DATA_BLOCK "DO_1_2_TON"   // DB244
{ S7_Optimized_Access := 'TRUE' }
AUTHOR : Simatic
FAMILY : IEC
NAME : IEC_TMR
VERSION : 1.0
// stored: InstanceOfName IEC_TIMER
"IEC_TIMER"
BEGIN
END_DATA_BLOCK

DATA_BLOCK "DO_2_0_TOF"   // DB246
{ S7_Optimized_Access := 'TRUE' }
AUTHOR : Simatic
FAMILY : IEC
NAME : IEC_TMR
VERSION : 1.0
// stored: InstanceOfName IEC_TIMER
"IEC_TIMER"
BEGIN
END_DATA_BLOCK

DATA_BLOCK "DO_1_2_TOF"   // DB247
{ S7_Optimized_Access := 'TRUE' }
AUTHOR : Simatic
FAMILY : IEC
NAME : IEC_TMR
VERSION : 1.0
// stored: InstanceOfName IEC_TIMER
"IEC_TIMER"
BEGIN
END_DATA_BLOCK

DATA_BLOCK "DI_1_1_TOF"   // DB253
{ S7_Optimized_Access := 'TRUE' }
AUTHOR : Simatic
FAMILY : IEC
NAME : IEC_TMR
VERSION : 1.0
// stored: InstanceOfName IEC_TIMER
"IEC_TIMER"
BEGIN
END_DATA_BLOCK

DATA_BLOCK "DI_1_4_TOF"   // DB255
{ S7_Optimized_Access := 'TRUE' }
AUTHOR : Simatic
FAMILY : IEC
NAME : IEC_TMR
VERSION : 1.0
// stored: InstanceOfName IEC_TIMER
"IEC_TIMER"
BEGIN
END_DATA_BLOCK

DATA_BLOCK "DI_1_11_TOF"   // DB256
{ S7_Optimized_Access := 'TRUE' }
AUTHOR : Simatic
FAMILY : IEC
NAME : IEC_TMR
VERSION : 1.0
// stored: InstanceOfName IEC_TIMER
"IEC_TIMER"
BEGIN
END_DATA_BLOCK

DATA_BLOCK "DO_1_4_TON"   // DB259
{ S7_Optimized_Access := 'TRUE' }
AUTHOR : Simatic
FAMILY : IEC
NAME : IEC_TMR
VERSION : 1.0
// stored: InstanceOfName IEC_TIMER
"IEC_TIMER"
BEGIN
END_DATA_BLOCK

DATA_BLOCK "DO_1_4_TOF"   // DB262
{ S7_Optimized_Access := 'TRUE' }
AUTHOR : Simatic
FAMILY : IEC
NAME : IEC_TMR
VERSION : 1.0
// stored: InstanceOfName IEC_TIMER
"IEC_TIMER"
BEGIN
END_DATA_BLOCK

DATA_BLOCK "DI_1_6_TOF"   // DB270
{ S7_Optimized_Access := 'TRUE' }
AUTHOR : Simatic
FAMILY : IEC
NAME : IEC_TMR
VERSION : 1.0
// stored: InstanceOfName IEC_TIMER
"IEC_TIMER"
BEGIN
END_DATA_BLOCK

DATA_BLOCK "DI_1_13_TOF"   // DB271
{ S7_Optimized_Access := 'TRUE' }
AUTHOR : Simatic
FAMILY : IEC
NAME : IEC_TMR
VERSION : 1.0
// stored: InstanceOfName IEC_TIMER
"IEC_TIMER"
BEGIN
END_DATA_BLOCK

DATA_BLOCK "DO_1_6_TON"   // DB274
{ S7_Optimized_Access := 'TRUE' }
AUTHOR : Simatic
FAMILY : IEC
NAME : IEC_TMR
VERSION : 1.0
// stored: InstanceOfName IEC_TIMER
"IEC_TIMER"
BEGIN
END_DATA_BLOCK

DATA_BLOCK "DO_1_6_TOF"   // DB277
{ S7_Optimized_Access := 'TRUE' }
AUTHOR : Simatic
FAMILY : IEC
NAME : IEC_TMR
VERSION : 1.0
// stored: InstanceOfName IEC_TIMER
"IEC_TIMER"
BEGIN
END_DATA_BLOCK

DATA_BLOCK "DI_1_2_TOF"   // DB285
{ S7_Optimized_Access := 'TRUE' }
AUTHOR : Simatic
FAMILY : IEC
NAME : IEC_TMR
VERSION : 1.0
// stored: InstanceOfName IEC_TIMER
"IEC_TIMER"
BEGIN
END_DATA_BLOCK

DATA_BLOCK "DI_1_5_TOF"   // DB287
{ S7_Optimized_Access := 'TRUE' }
AUTHOR : Simatic
FAMILY : IEC
NAME : IEC_TMR
VERSION : 1.0
// stored: InstanceOfName IEC_TIMER
"IEC_TIMER"
BEGIN
END_DATA_BLOCK

DATA_BLOCK "DI_1_12_TOF"   // DB288
{ S7_Optimized_Access := 'TRUE' }
AUTHOR : Simatic
FAMILY : IEC
NAME : IEC_TMR
VERSION : 1.0
// stored: InstanceOfName IEC_TIMER
"IEC_TIMER"
BEGIN
END_DATA_BLOCK

DATA_BLOCK "DO_1_5_TON"   // DB291
{ S7_Optimized_Access := 'TRUE' }
AUTHOR : Simatic
FAMILY : IEC
NAME : IEC_TMR
VERSION : 1.0
// stored: InstanceOfName IEC_TIMER
"IEC_TIMER"
BEGIN
END_DATA_BLOCK

DATA_BLOCK "DO_1_5_TOF"   // DB294
{ S7_Optimized_Access := 'TRUE' }
AUTHOR : Simatic
FAMILY : IEC
NAME : IEC_TMR
VERSION : 1.0
// stored: InstanceOfName IEC_TIMER
"IEC_TIMER"
BEGIN
END_DATA_BLOCK

// folder: (top level)

FUNCTION "Valve" : Void   // FC1, SCL
{ S7_Optimized_Access := 'TRUE' }
VERSION : 0.1
   VAR_INPUT
      Valve_opening : Bool;
      Need_open : Bool;
   END_VAR
   VAR_OUTPUT
      CMD_Open_Out : Bool;
      Alarm_Out : Bool;
   END_VAR
   VAR_IN_OUT
      valve : Struct
         CMD_Open : Bool;   // Команда открыть
         CMD_Close : Bool;   // Команда закрыть
         CMD_ALRM_Stop : Bool;
         State : Word;
         State_INT : Int;
         Mode : Bool;   // 0-ручной, 1-авто
         Alarm : Word;
         bools : Word;
         RST_ALRM : Bool;
         CMD_Open_Out : Bool;   // управление открыть
         CMD_Close_Out : Bool;   // управление закрыть
      END_STRUCT;
      TIME_Opening : TON_TIME;
      TIME_Closing : TON_TIME;
   END_VAR
BEGIN
   IF (#valve.Alarm = 0) AND #Need_open
   THEN
       #valve.CMD_Open := 1;
   ELSE
       #valve.CMD_Open := 0;
   END_IF;


   IF #valve.Alarm = 0
   THEN
      #valve.CMD_Open_Out := #valve.CMD_Open;

   ELSE
      #valve.CMD_Open_Out := FALSE;

   END_IF;

   //формирование состояний
   (*#valve.State.%X3 := #Valve_opening;
   #valve.State.%X4 := NOT (#Valve_opening);*)

   IF #valve.Alarm.%X1 THEN
       #valve.State := 1;
   END_IF;
   IF #valve.Alarm.%X2 THEN
       #valve.State := 2;
   END_IF;
   IF #Valve_opening AND NOT (#valve.Alarm.%X1 OR #valve.Alarm.%X2) THEN
       #valve.State := 3;
   END_IF;
   IF NOT (#Valve_opening) AND NOT (#valve.Alarm.%X1 OR #valve.Alarm.%X2) THEN
       #valve.State := 4;
   END_IF;

   //аварии при открытии и закрытии
   #TIME_Opening.TON(IN := #valve.CMD_Open_Out AND NOT (#Valve_opening),
   PT := T#25s);
   IF #TIME_Opening.Q THEN
       #valve.Alarm.%X1 := TRUE;
   END_IF;
   (*#valve.State.%X1 := #valve.Alarm.%X1;*)

   #TIME_Closing.TON(IN := NOT #valve.CMD_Open_Out AND #Valve_opening,
   PT := T#25s);
   IF #TIME_Closing.Q THEN
       #valve.Alarm.%X2 := TRUE;
   END_IF;
   (*#valve.State.%X2 := #valve.Alarm.%X2;*)

   IF #valve.RST_ALRM THEN
       #valve.Alarm := 0;
       #valve.RST_ALRM := 0;
   END_IF;



   #CMD_Open_Out := #valve.CMD_Open_Out;

   IF #valve.Alarm <> 0
   THEN
       #Alarm_Out := 1;
   END_IF;
END_FUNCTION

FUNCTION "DI" : Void   // FC2, LAD
{ S7_Optimized_Access := 'TRUE' }
VERSION : 0.1
   VAR_INPUT
      Input : Bool;   // Входной сигнал
   END_VAR
   VAR_IN_OUT
      DI : Struct
         Time_ON : Int;   // Время перехода OFF->ON
         Time_OFF : Int;   // Время перехода ON->OFF
         Input : Bool;   // Значение с модуля
         Disable : Bool;   // Запрет обработки канала
         Invert : Bool;   // Инертирование канала
         Output : Bool;   // Значение канала для логики
      END_STRUCT;
      TON_Timer : IEC_TIMER;
      TOF_Timer : IEC_TIMER;
   END_VAR
   VAR_TEMP
      Time_ON_int : Time;
      Time_OFF_int : Time;
      et1 : Time;
      et2 : Time;
      trig_et : Bool;
   END_VAR
BEGIN

REGION Network 1: Конверация времени
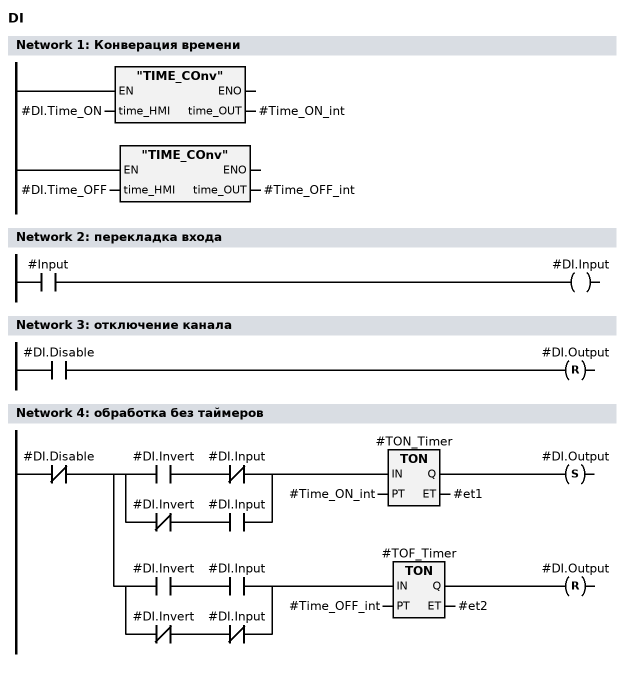
   RUNG wire#powerrail
      "TIME_COnv"(time_HMI := #DI.Time_ON, time_OUT => #Time_ON_int)
   END_RUNG
   RUNG wire#powerrail
      "TIME_COnv"(time_HMI := #DI.Time_OFF, time_OUT => #Time_OFF_int)
   END_RUNG
   // the same network as SCL:
   "TIME_COnv"(time_HMI := #DI.Time_ON, time_OUT => #Time_ON_int);
   "TIME_COnv"(time_HMI := #DI.Time_OFF, time_OUT => #Time_OFF_int);
END_REGION

REGION Network 2: перекладка входа
   RUNG wire#powerrail
      Contact( #Input )
      Coil( #DI.Input )
   END_RUNG
   // the same network as SCL:
   #DI.Input := #Input;
END_REGION

REGION Network 3: отключение канала
   RUNG wire#powerrail
      Contact( #DI.Disable )
      R_Coil( #DI.Output )
   END_RUNG
   // the same network as SCL:
   IF #DI.Disable THEN #DI.Output := FALSE; END_IF;
END_REGION

REGION Network 4: обработка без таймеров
   #TON_Timer.TON(IN := NOT #DI.Disable AND ((#DI.Invert AND NOT #DI.Input) OR (NOT #DI.Invert AND #DI.Input)),
                  PT := #Time_ON_int,
                  ET => #et1);
   IF #TON_Timer.Q THEN #DI.Output := TRUE; END_IF;
   #TOF_Timer.TON(IN := NOT #DI.Disable AND ((#DI.Invert AND #DI.Input) OR (NOT #DI.Invert AND NOT #DI.Input)),
                  PT := #Time_OFF_int,
                  ET => #et2);
   IF #TOF_Timer.Q THEN #DI.Output := FALSE; END_IF;
END_REGION
END_FUNCTION

FUNCTION "DO" : Void   // FC3, LAD
{ S7_Optimized_Access := 'TRUE' }
VERSION : 0.1
   VAR_OUTPUT
      Output : Bool;
   END_VAR
   VAR_IN_OUT
      "DO" : Struct
         Time_ON : Int;   // Время перехода OFF->ON
         Time_OFF : Int;   // Время перехода ON->OFF
         Input : Bool;   // Значение от логики
         Disable : Bool;   // Запрет обработки канала
         Invert : Bool;   // Инертирование канала
         Output : Bool;   // Значение на модуль
      END_STRUCT;
      TON_Timer : IEC_TIMER;
      TOF_Timer : IEC_TIMER;
   END_VAR
   VAR_TEMP
      Time_ON_int : Time;
      Time_OFF_int : Time;
      et1 : Time;
      et2 : Time;
   END_VAR
BEGIN

REGION Network 1: Конверация времени
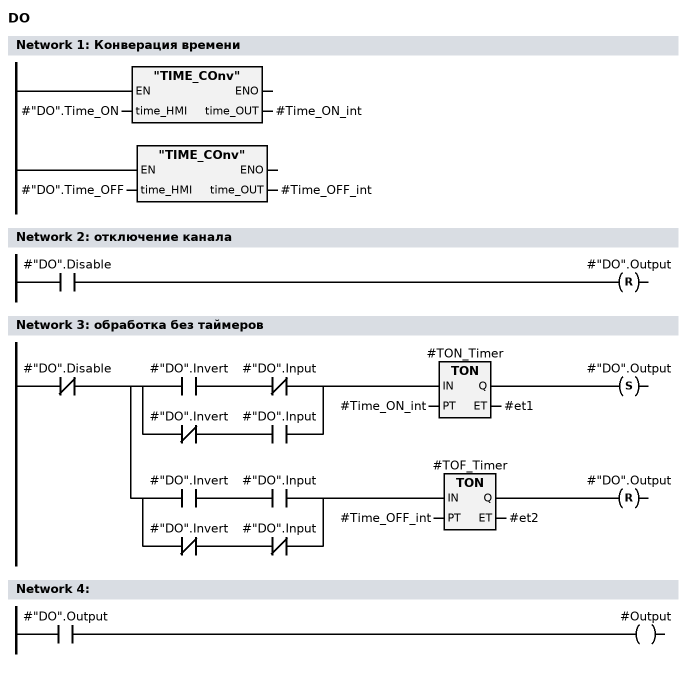
   RUNG wire#powerrail
      "TIME_COnv"(time_HMI := #"DO".Time_ON, time_OUT => #Time_ON_int)
   END_RUNG
   RUNG wire#powerrail
      "TIME_COnv"(time_HMI := #"DO".Time_OFF, time_OUT => #Time_OFF_int)
   END_RUNG
   // the same network as SCL:
   "TIME_COnv"(time_HMI := #"DO".Time_ON, time_OUT => #Time_ON_int);
   "TIME_COnv"(time_HMI := #"DO".Time_OFF, time_OUT => #Time_OFF_int);
END_REGION

REGION Network 2: отключение канала
   RUNG wire#powerrail
      Contact( #"DO".Disable )
      R_Coil( #"DO".Output )
   END_RUNG
   // the same network as SCL:
   IF #"DO".Disable THEN #"DO".Output := FALSE; END_IF;
END_REGION

REGION Network 3: обработка без таймеров
   #TON_Timer.TON(IN := NOT #"DO".Disable AND ((#"DO".Invert AND NOT #"DO".Input) OR (NOT #"DO".Invert AND #"DO".Input)),
                  PT := #Time_ON_int,
                  ET => #et1);
   IF #TON_Timer.Q THEN #"DO".Output := TRUE; END_IF;
   #TOF_Timer.TON(IN := NOT #"DO".Disable AND ((#"DO".Invert AND #"DO".Input) OR (NOT #"DO".Invert AND NOT #"DO".Input)),
                  PT := #Time_OFF_int,
                  ET => #et2);
   IF #TOF_Timer.Q THEN #"DO".Output := FALSE; END_IF;
END_REGION

REGION Network 4
   RUNG wire#powerrail
      Contact( #"DO".Output )
      Coil( #Output )
   END_RUNG
   // the same network as SCL:
   #Output := #"DO".Output;
END_REGION
END_FUNCTION

FUNCTION "Gaz" : Void   // FC4, SCL
{ S7_Optimized_Access := 'TRUE' }
VERSION : 0.1
BEGIN
   IF "PLC_Signals_DB".AI_2_6.State.%X1 THEN
       "DB_TST".Gaz_state := 2;
       ELSE 
           IF "PLC_Signals_DB".AI_2_6.State.%X2 THEN
               "DB_TST".Gaz_state := 1;
           ELSE
               "DB_TST".Gaz_state := 0;
           END_IF;
   END_IF;
END_FUNCTION

FUNCTION "AI_CONV" : Void   // FC6, SCL
{ S7_Optimized_Access := 'TRUE' }
VERSION : 0.1
   VAR_IN_OUT
      AI : Struct   // Структура AI
         Hihi_Value : Real;   // True
         High_Value : Real;   // True
         Low_Value : Real;   // True
         Lolo_Value : Real;   // True
         MIN_Current : Real;   // True
         MAX_Current : Real;   // True
         MAX_Value : Real;   // True
         MIN_Value : Real;   // True
         Underflow_RAW : Real;   // True
         Overflow_RAW : Real;   // True
         SCALED : Real;   // True
         ING_Value : Real;   // True
         Manual_Value : Real;   // True
         Alarm_Delay : Int;   // True
         Warning_Delay : Int;   // True
         AVG_Delay : Real;   // True
         Underflow_Delay : Int;   // True
         Overflow_Delay : Int;   // True
         State : Word;   // True
         Modeee : Word;   // True
         bools : Word;   // True
         AI_RAW_MIN : Int;   // True
         AI_RAW_MAX : Int;   // True
         Hihi_EN : Bool;   // True
         High_EN : Bool;   // True
         Low_En : Bool;   // True
         Lolo_EN : Bool;   // True
      END_STRUCT;
      AI_RAW : Int;   // ???????? ??? ?? ?????
      Hihi_TImer : TON_TIME;
      High_Timer : TON_TIME;
      Low_Timer : TON_TIME;
      Lolo_Timer : TON_TIME;
      WB_Timer : TON_TIME;
      OVerflow_Timer : TON_TIME;
   END_VAR
BEGIN
   (*
   #AI.mA := (#AI.ACP - #AI.ACP_LO) * ((#AI.mA_HI - #AI.mA_LO) / (#AI.ACP_HI - #AI.ACP_LO)) + #AI.mA_LO;
   #AI.ENG := (#AI.mA - #AI.mA_LO) * ((#AI.ENG_HI - #AI.ENG_LO) / (#AI.mA_HI - #AI.mA_LO)) + #AI.ENG_LO;
   *)
   //IF #AI.Modeee.%X0 THEN
       #AI.ING_Value := (#AI_RAW - #AI.AI_RAW_MIN) * ((#AI.MAX_Current - #AI.MIN_Current) / (#AI.AI_RAW_MAX - #AI.AI_RAW_MIN)) + #AI.MIN_Current;
       #AI.SCALED := (#AI_RAW - #AI.AI_RAW_MIN) * ((#AI.MAX_Value - #AI.MIN_Value) / (#AI.AI_RAW_MAX - #AI.AI_RAW_MIN)) + #AI.MIN_Value;




   //END_IF;


   (* #AI.mA := (#AI.ACP - #AI.ACP_LO) * ((#AI.mA_HI - #AI.mA_LO) / (#AI.ACP_HI - #AI.ACP_LO)) + #AI.mA_LO;
   #AI.ENG := (#AI.mA - #AI.mA_LO) * ((#AI.ENG_HI - #AI.ENG_LO) / (#AI.mA_HI - #AI.mA_LO)) + #AI.ENG_LO;

   IF NOT #AI.Repair THEN
       #AI.State_W.%X7 := FALSE;
       IF #AI.ENG <= #AI.ENG_Set_LoLo THEN
           #AI.LoLo := TRUE;
           #AI.State_W.%X0 := TRUE;
       ELSE
           #AI.LoLo := FALSE;
           #AI.State_W.%X0 := FALSE;
       END_IF;

       IF #AI.ENG <= #AI.ENG_Set_Lo THEN
           #AI.Lo := TRUE;
           #AI.State_W.%X1 := TRUE;
       ELSE
           #AI.Lo := FALSE;
           #AI.State_W.%X1 := FALSE;
       END_IF;

       IF #AI.ENG >= #AI.ENG_Set_Hi THEN
           #AI.Hi := TRUE;
           #AI.State_W.%X2 := TRUE;
       ELSE
           #AI.Hi := FALSE;
           #AI.State_W.%X2 := FALSE;
       END_IF;

       IF #AI.ENG >= #AI.ENG_Set_HiHi THEN
           #AI.HiHi := TRUE;
           #AI.State_W.%X3 := TRUE;
       ELSE
           #AI.HiHi := FALSE;
           #AI.State_W.%X3 := FALSE;
       END_IF;

       IF #AI.mA <= 3.5 THEN
           #AI.BL := TRUE;
           #AI.State_W.%X4 := TRUE;
       ELSE
           #AI.BL := FALSE;
           #AI.State_W.%X4 := FALSE;
       END_IF;

       IF #AI.mA >= 20.5 THEN
           #AI.OL := TRUE;
           #AI.State_W.%X5 := TRUE;
       ELSE
           #AI.OL := FALSE;
           #AI.State_W.%X5 := FALSE;
       END_IF;

       #AI.State_W.%X6 := #AI.State_W.%X4 OR #AI.State_W.%X5;

       IF #AI.OL OR #AI.BL THEN
           #AI.State := 3;
       ELSIF #AI.HiHi OR #AI.LoLo THEN
           #AI.State := 2;
       ELSIF #AI.Hi OR #AI.Lo THEN
           #AI.State := 1;
       ELSE
           #AI.State := 0;
       END_IF;

   ELSE
       #AI.LoLo := FALSE; #AI.Lo := FALSE; #AI.Hi := FALSE; #AI.HiHi := FALSE;
       #AI.OL := FALSE; #AI.BL := FALSE;
       #AI.State := 4;
       #AI.State_W := 0;
       #AI.State_W.%X7 := TRUE;
   END_IF;
   #AI.Mode := #AI.Repair; *)
END_FUNCTION

FUNCTION "AI_TST" : Void   // FC7, LAD
{ S7_Optimized_Access := 'TRUE' }
VERSION : 0.1
BEGIN

REGION Network 1: Давление на выходе, МПа
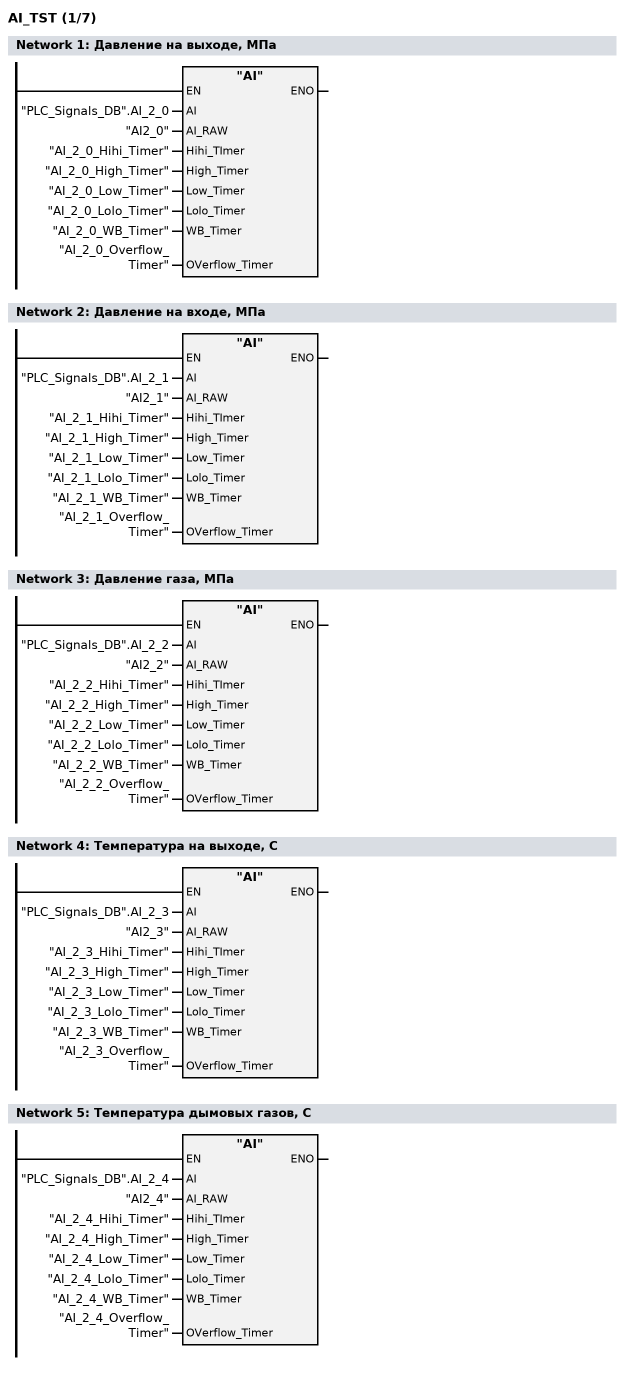
   RUNG wire#powerrail
      "AI"(AI := "PLC_Signals_DB".AI_2_0, AI_RAW := "AI2_0", Hihi_TImer := "AI_2_0_Hihi_Timer", High_Timer := "AI_2_0_High_Timer", Low_Timer := "AI_2_0_Low_Timer", Lolo_Timer := "AI_2_0_Lolo_Timer", WB_Timer := "AI_2_0_WB_Timer", OVerflow_Timer := "AI_2_0_Overflow_Timer")
   END_RUNG
   // the same network as SCL:
   "AI"(AI := "PLC_Signals_DB".AI_2_0,
        AI_RAW := "AI2_0",
        Hihi_TImer := "AI_2_0_Hihi_Timer",
        High_Timer := "AI_2_0_High_Timer",
        Low_Timer := "AI_2_0_Low_Timer",
        Lolo_Timer := "AI_2_0_Lolo_Timer",
        WB_Timer := "AI_2_0_WB_Timer",
        OVerflow_Timer := "AI_2_0_Overflow_Timer");
END_REGION

REGION Network 2: Давление на входе, МПа
   RUNG wire#powerrail
      "AI"(AI := "PLC_Signals_DB".AI_2_1, AI_RAW := "AI2_1", Hihi_TImer := "AI_2_1_Hihi_Timer", High_Timer := "AI_2_1_High_Timer", Low_Timer := "AI_2_1_Low_Timer", Lolo_Timer := "AI_2_1_Lolo_Timer", WB_Timer := "AI_2_1_WB_Timer", OVerflow_Timer := "AI_2_1_Overflow_Timer")
   END_RUNG
   // the same network as SCL:
   "AI"(AI := "PLC_Signals_DB".AI_2_1,
        AI_RAW := "AI2_1",
        Hihi_TImer := "AI_2_1_Hihi_Timer",
        High_Timer := "AI_2_1_High_Timer",
        Low_Timer := "AI_2_1_Low_Timer",
        Lolo_Timer := "AI_2_1_Lolo_Timer",
        WB_Timer := "AI_2_1_WB_Timer",
        OVerflow_Timer := "AI_2_1_Overflow_Timer");
END_REGION

REGION Network 3: Давление газа, МПа
   RUNG wire#powerrail
      "AI"(AI := "PLC_Signals_DB".AI_2_2, AI_RAW := "AI2_2", Hihi_TImer := "AI_2_2_Hihi_Timer", High_Timer := "AI_2_2_High_Timer", Low_Timer := "AI_2_2_Low_Timer", Lolo_Timer := "AI_2_2_Lolo_Timer", WB_Timer := "AI_2_2_WB_Timer", OVerflow_Timer := "AI_2_2_Overflow_Timer")
   END_RUNG
   // the same network as SCL:
   "AI"(AI := "PLC_Signals_DB".AI_2_2,
        AI_RAW := "AI2_2",
        Hihi_TImer := "AI_2_2_Hihi_Timer",
        High_Timer := "AI_2_2_High_Timer",
        Low_Timer := "AI_2_2_Low_Timer",
        Lolo_Timer := "AI_2_2_Lolo_Timer",
        WB_Timer := "AI_2_2_WB_Timer",
        OVerflow_Timer := "AI_2_2_Overflow_Timer");
END_REGION

REGION Network 4: Температура на выходе, С
   RUNG wire#powerrail
      "AI"(AI := "PLC_Signals_DB".AI_2_3, AI_RAW := "AI2_3", Hihi_TImer := "AI_2_3_Hihi_Timer", High_Timer := "AI_2_3_High_Timer", Low_Timer := "AI_2_3_Low_Timer", Lolo_Timer := "AI_2_3_Lolo_Timer", WB_Timer := "AI_2_3_WB_Timer", OVerflow_Timer := "AI_2_3_Overflow_Timer")
   END_RUNG
   // the same network as SCL:
   "AI"(AI := "PLC_Signals_DB".AI_2_3,
        AI_RAW := "AI2_3",
        Hihi_TImer := "AI_2_3_Hihi_Timer",
        High_Timer := "AI_2_3_High_Timer",
        Low_Timer := "AI_2_3_Low_Timer",
        Lolo_Timer := "AI_2_3_Lolo_Timer",
        WB_Timer := "AI_2_3_WB_Timer",
        OVerflow_Timer := "AI_2_3_Overflow_Timer");
END_REGION

REGION Network 5: Температура дымовых газов, С
   RUNG wire#powerrail
      "AI"(AI := "PLC_Signals_DB".AI_2_4, AI_RAW := "AI2_4", Hihi_TImer := "AI_2_4_Hihi_Timer", High_Timer := "AI_2_4_High_Timer", Low_Timer := "AI_2_4_Low_Timer", Lolo_Timer := "AI_2_4_Lolo_Timer", WB_Timer := "AI_2_4_WB_Timer", OVerflow_Timer := "AI_2_4_Overflow_Timer")
   END_RUNG
   // the same network as SCL:
   "AI"(AI := "PLC_Signals_DB".AI_2_4,
        AI_RAW := "AI2_4",
        Hihi_TImer := "AI_2_4_Hihi_Timer",
        High_Timer := "AI_2_4_High_Timer",
        Low_Timer := "AI_2_4_Low_Timer",
        Lolo_Timer := "AI_2_4_Lolo_Timer",
        WB_Timer := "AI_2_4_WB_Timer",
        OVerflow_Timer := "AI_2_4_Overflow_Timer");
END_REGION

REGION Network 6: Температура ёмкости, С
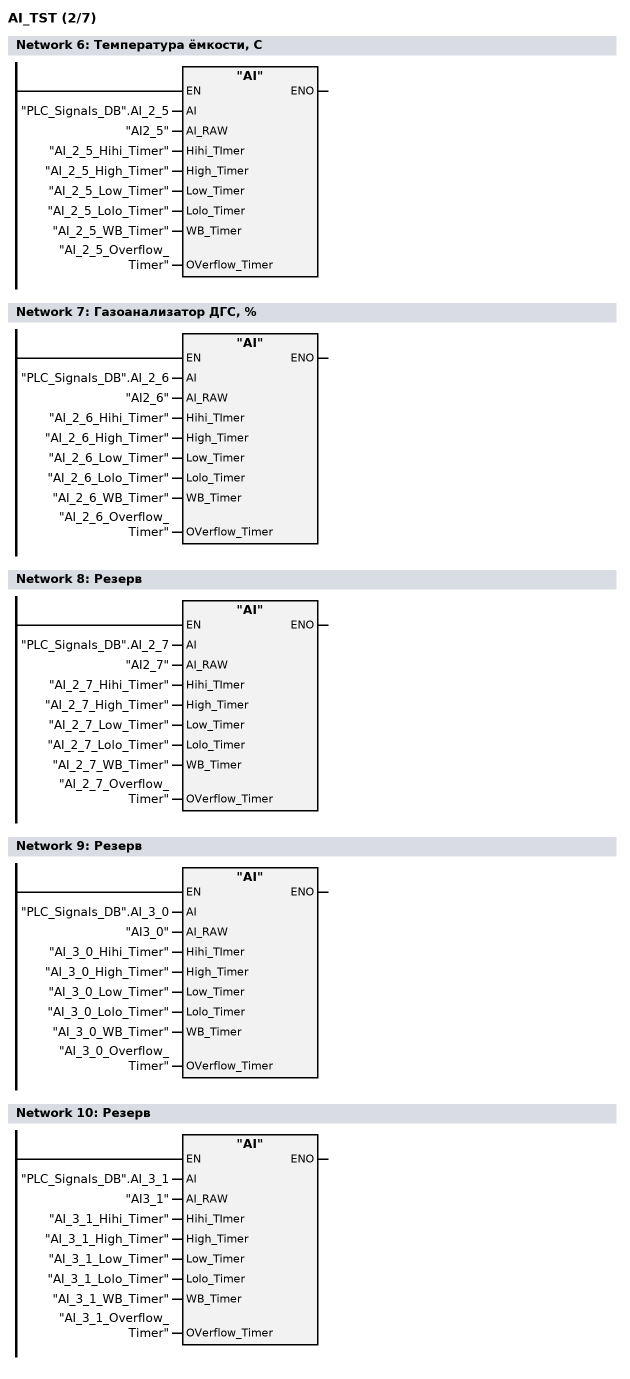
   RUNG wire#powerrail
      "AI"(AI := "PLC_Signals_DB".AI_2_5, AI_RAW := "AI2_5", Hihi_TImer := "AI_2_5_Hihi_Timer", High_Timer := "AI_2_5_High_Timer", Low_Timer := "AI_2_5_Low_Timer", Lolo_Timer := "AI_2_5_Lolo_Timer", WB_Timer := "AI_2_5_WB_Timer", OVerflow_Timer := "AI_2_5_Overflow_Timer")
   END_RUNG
   // the same network as SCL:
   "AI"(AI := "PLC_Signals_DB".AI_2_5,
        AI_RAW := "AI2_5",
        Hihi_TImer := "AI_2_5_Hihi_Timer",
        High_Timer := "AI_2_5_High_Timer",
        Low_Timer := "AI_2_5_Low_Timer",
        Lolo_Timer := "AI_2_5_Lolo_Timer",
        WB_Timer := "AI_2_5_WB_Timer",
        OVerflow_Timer := "AI_2_5_Overflow_Timer");
END_REGION

REGION Network 7: Газоанализатор ДГС, %
   RUNG wire#powerrail
      "AI"(AI := "PLC_Signals_DB".AI_2_6, AI_RAW := "AI2_6", Hihi_TImer := "AI_2_6_Hihi_Timer", High_Timer := "AI_2_6_High_Timer", Low_Timer := "AI_2_6_Low_Timer", Lolo_Timer := "AI_2_6_Lolo_Timer", WB_Timer := "AI_2_6_WB_Timer", OVerflow_Timer := "AI_2_6_Overflow_Timer")
   END_RUNG
   // the same network as SCL:
   "AI"(AI := "PLC_Signals_DB".AI_2_6,
        AI_RAW := "AI2_6",
        Hihi_TImer := "AI_2_6_Hihi_Timer",
        High_Timer := "AI_2_6_High_Timer",
        Low_Timer := "AI_2_6_Low_Timer",
        Lolo_Timer := "AI_2_6_Lolo_Timer",
        WB_Timer := "AI_2_6_WB_Timer",
        OVerflow_Timer := "AI_2_6_Overflow_Timer");
END_REGION

REGION Network 8: Резерв
   RUNG wire#powerrail
      "AI"(AI := "PLC_Signals_DB".AI_2_7, AI_RAW := "AI2_7", Hihi_TImer := "AI_2_7_Hihi_Timer", High_Timer := "AI_2_7_High_Timer", Low_Timer := "AI_2_7_Low_Timer", Lolo_Timer := "AI_2_7_Lolo_Timer", WB_Timer := "AI_2_7_WB_Timer", OVerflow_Timer := "AI_2_7_Overflow_Timer")
   END_RUNG
   // the same network as SCL:
   "AI"(AI := "PLC_Signals_DB".AI_2_7,
        AI_RAW := "AI2_7",
        Hihi_TImer := "AI_2_7_Hihi_Timer",
        High_Timer := "AI_2_7_High_Timer",
        Low_Timer := "AI_2_7_Low_Timer",
        Lolo_Timer := "AI_2_7_Lolo_Timer",
        WB_Timer := "AI_2_7_WB_Timer",
        OVerflow_Timer := "AI_2_7_Overflow_Timer");
END_REGION

REGION Network 9: Резерв
   RUNG wire#powerrail
      "AI"(AI := "PLC_Signals_DB".AI_3_0, AI_RAW := "AI3_0", Hihi_TImer := "AI_3_0_Hihi_Timer", High_Timer := "AI_3_0_High_Timer", Low_Timer := "AI_3_0_Low_Timer", Lolo_Timer := "AI_3_0_Lolo_Timer", WB_Timer := "AI_3_0_WB_Timer", OVerflow_Timer := "AI_3_0_Overflow_Timer")
   END_RUNG
   // the same network as SCL:
   "AI"(AI := "PLC_Signals_DB".AI_3_0,
        AI_RAW := "AI3_0",
        Hihi_TImer := "AI_3_0_Hihi_Timer",
        High_Timer := "AI_3_0_High_Timer",
        Low_Timer := "AI_3_0_Low_Timer",
        Lolo_Timer := "AI_3_0_Lolo_Timer",
        WB_Timer := "AI_3_0_WB_Timer",
        OVerflow_Timer := "AI_3_0_Overflow_Timer");
END_REGION

REGION Network 10: Резерв
   RUNG wire#powerrail
      "AI"(AI := "PLC_Signals_DB".AI_3_1, AI_RAW := "AI3_1", Hihi_TImer := "AI_3_1_Hihi_Timer", High_Timer := "AI_3_1_High_Timer", Low_Timer := "AI_3_1_Low_Timer", Lolo_Timer := "AI_3_1_Lolo_Timer", WB_Timer := "AI_3_1_WB_Timer", OVerflow_Timer := "AI_3_1_Overflow_Timer")
   END_RUNG
   // the same network as SCL:
   "AI"(AI := "PLC_Signals_DB".AI_3_1,
        AI_RAW := "AI3_1",
        Hihi_TImer := "AI_3_1_Hihi_Timer",
        High_Timer := "AI_3_1_High_Timer",
        Low_Timer := "AI_3_1_Low_Timer",
        Lolo_Timer := "AI_3_1_Lolo_Timer",
        WB_Timer := "AI_3_1_WB_Timer",
        OVerflow_Timer := "AI_3_1_Overflow_Timer");
END_REGION

REGION Network 11: Резерв
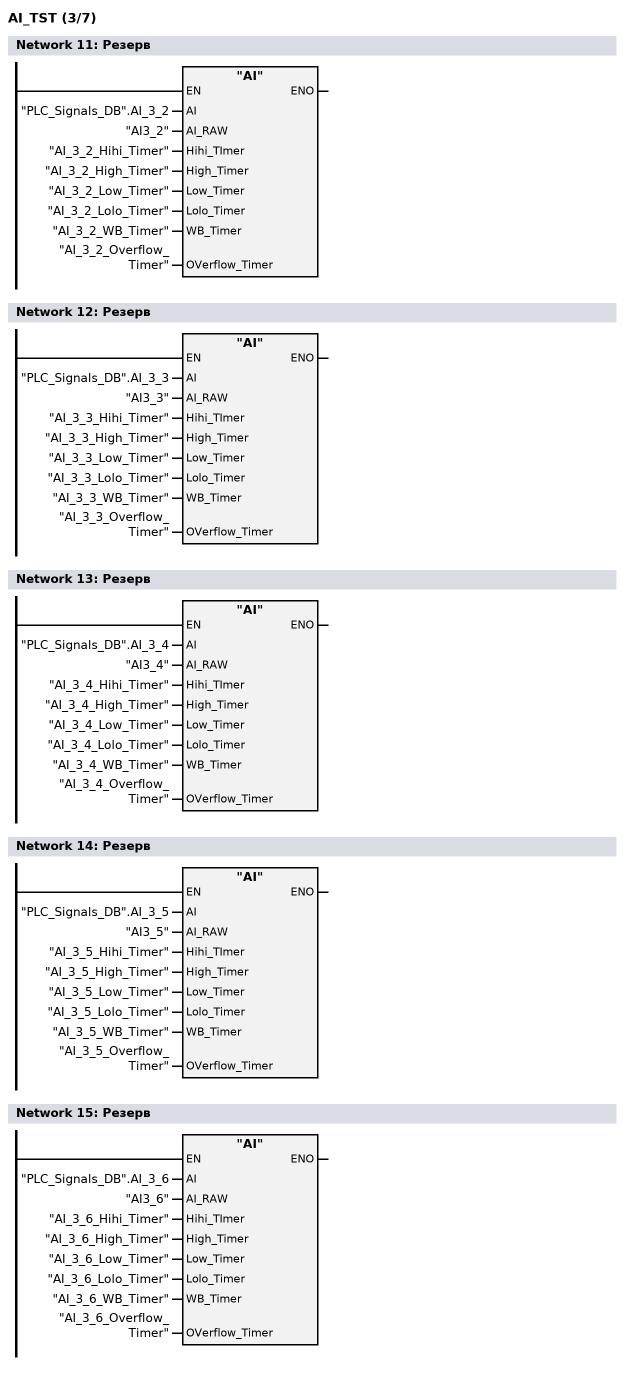
   RUNG wire#powerrail
      "AI"(AI := "PLC_Signals_DB".AI_3_2, AI_RAW := "AI3_2", Hihi_TImer := "AI_3_2_Hihi_Timer", High_Timer := "AI_3_2_High_Timer", Low_Timer := "AI_3_2_Low_Timer", Lolo_Timer := "AI_3_2_Lolo_Timer", WB_Timer := "AI_3_2_WB_Timer", OVerflow_Timer := "AI_3_2_Overflow_Timer")
   END_RUNG
   // the same network as SCL:
   "AI"(AI := "PLC_Signals_DB".AI_3_2,
        AI_RAW := "AI3_2",
        Hihi_TImer := "AI_3_2_Hihi_Timer",
        High_Timer := "AI_3_2_High_Timer",
        Low_Timer := "AI_3_2_Low_Timer",
        Lolo_Timer := "AI_3_2_Lolo_Timer",
        WB_Timer := "AI_3_2_WB_Timer",
        OVerflow_Timer := "AI_3_2_Overflow_Timer");
END_REGION

REGION Network 12: Резерв
   RUNG wire#powerrail
      "AI"(AI := "PLC_Signals_DB".AI_3_3, AI_RAW := "AI3_3", Hihi_TImer := "AI_3_3_Hihi_Timer", High_Timer := "AI_3_3_High_Timer", Low_Timer := "AI_3_3_Low_Timer", Lolo_Timer := "AI_3_3_Lolo_Timer", WB_Timer := "AI_3_3_WB_Timer", OVerflow_Timer := "AI_3_3_Overflow_Timer")
   END_RUNG
   // the same network as SCL:
   "AI"(AI := "PLC_Signals_DB".AI_3_3,
        AI_RAW := "AI3_3",
        Hihi_TImer := "AI_3_3_Hihi_Timer",
        High_Timer := "AI_3_3_High_Timer",
        Low_Timer := "AI_3_3_Low_Timer",
        Lolo_Timer := "AI_3_3_Lolo_Timer",
        WB_Timer := "AI_3_3_WB_Timer",
        OVerflow_Timer := "AI_3_3_Overflow_Timer");
END_REGION

REGION Network 13: Резерв
   RUNG wire#powerrail
      "AI"(AI := "PLC_Signals_DB".AI_3_4, AI_RAW := "AI3_4", Hihi_TImer := "AI_3_4_Hihi_Timer", High_Timer := "AI_3_4_High_Timer", Low_Timer := "AI_3_4_Low_Timer", Lolo_Timer := "AI_3_4_Lolo_Timer", WB_Timer := "AI_3_4_WB_Timer", OVerflow_Timer := "AI_3_4_Overflow_Timer")
   END_RUNG
   // the same network as SCL:
   "AI"(AI := "PLC_Signals_DB".AI_3_4,
        AI_RAW := "AI3_4",
        Hihi_TImer := "AI_3_4_Hihi_Timer",
        High_Timer := "AI_3_4_High_Timer",
        Low_Timer := "AI_3_4_Low_Timer",
        Lolo_Timer := "AI_3_4_Lolo_Timer",
        WB_Timer := "AI_3_4_WB_Timer",
        OVerflow_Timer := "AI_3_4_Overflow_Timer");
END_REGION

REGION Network 14: Резерв
   RUNG wire#powerrail
      "AI"(AI := "PLC_Signals_DB".AI_3_5, AI_RAW := "AI3_5", Hihi_TImer := "AI_3_5_Hihi_Timer", High_Timer := "AI_3_5_High_Timer", Low_Timer := "AI_3_5_Low_Timer", Lolo_Timer := "AI_3_5_Lolo_Timer", WB_Timer := "AI_3_5_WB_Timer", OVerflow_Timer := "AI_3_5_Overflow_Timer")
   END_RUNG
   // the same network as SCL:
   "AI"(AI := "PLC_Signals_DB".AI_3_5,
        AI_RAW := "AI3_5",
        Hihi_TImer := "AI_3_5_Hihi_Timer",
        High_Timer := "AI_3_5_High_Timer",
        Low_Timer := "AI_3_5_Low_Timer",
        Lolo_Timer := "AI_3_5_Lolo_Timer",
        WB_Timer := "AI_3_5_WB_Timer",
        OVerflow_Timer := "AI_3_5_Overflow_Timer");
END_REGION

REGION Network 15: Резерв
   RUNG wire#powerrail
      "AI"(AI := "PLC_Signals_DB".AI_3_6, AI_RAW := "AI3_6", Hihi_TImer := "AI_3_6_Hihi_Timer", High_Timer := "AI_3_6_High_Timer", Low_Timer := "AI_3_6_Low_Timer", Lolo_Timer := "AI_3_6_Lolo_Timer", WB_Timer := "AI_3_6_WB_Timer", OVerflow_Timer := "AI_3_6_Overflow_Timer")
   END_RUNG
   // the same network as SCL:
   "AI"(AI := "PLC_Signals_DB".AI_3_6,
        AI_RAW := "AI3_6",
        Hihi_TImer := "AI_3_6_Hihi_Timer",
        High_Timer := "AI_3_6_High_Timer",
        Low_Timer := "AI_3_6_Low_Timer",
        Lolo_Timer := "AI_3_6_Lolo_Timer",
        WB_Timer := "AI_3_6_WB_Timer",
        OVerflow_Timer := "AI_3_6_Overflow_Timer");
END_REGION

REGION Network 16: Резерв
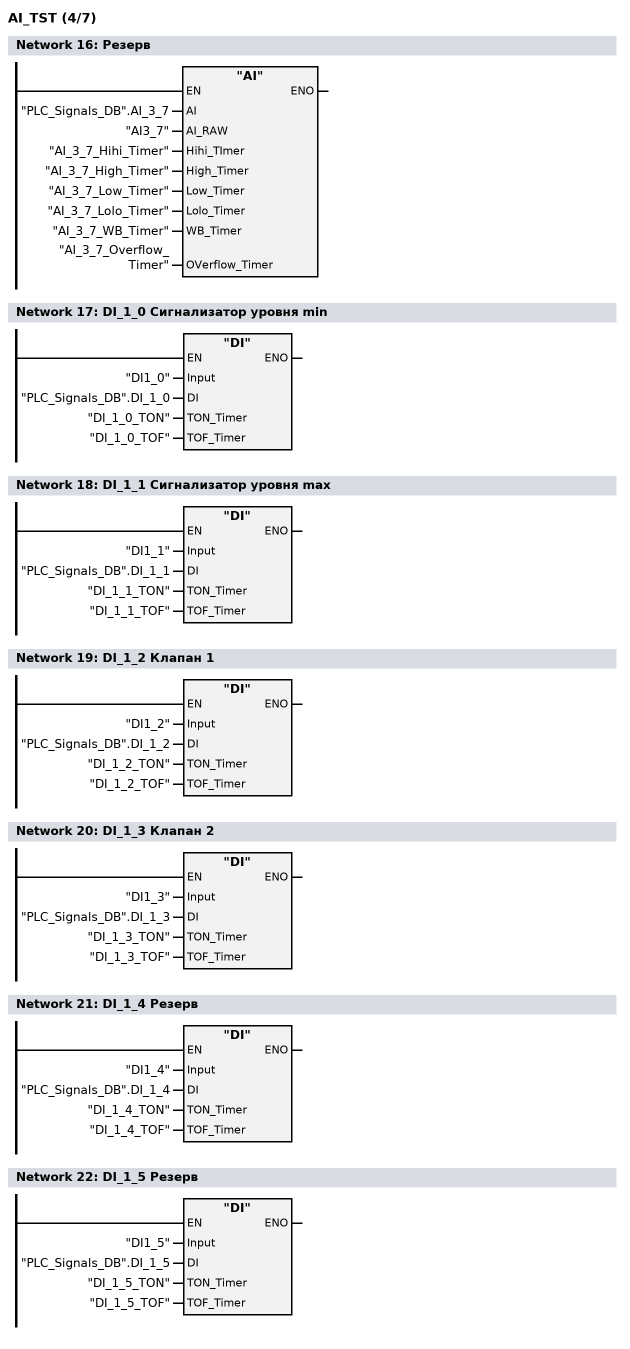
   RUNG wire#powerrail
      "AI"(AI := "PLC_Signals_DB".AI_3_7, AI_RAW := "AI3_7", Hihi_TImer := "AI_3_7_Hihi_Timer", High_Timer := "AI_3_7_High_Timer", Low_Timer := "AI_3_7_Low_Timer", Lolo_Timer := "AI_3_7_Lolo_Timer", WB_Timer := "AI_3_7_WB_Timer", OVerflow_Timer := "AI_3_7_Overflow_Timer")
   END_RUNG
   // the same network as SCL:
   "AI"(AI := "PLC_Signals_DB".AI_3_7,
        AI_RAW := "AI3_7",
        Hihi_TImer := "AI_3_7_Hihi_Timer",
        High_Timer := "AI_3_7_High_Timer",
        Low_Timer := "AI_3_7_Low_Timer",
        Lolo_Timer := "AI_3_7_Lolo_Timer",
        WB_Timer := "AI_3_7_WB_Timer",
        OVerflow_Timer := "AI_3_7_Overflow_Timer");
END_REGION

REGION Network 17: DI_1_0 Сигнализатор уровня min
   RUNG wire#powerrail
      "DI"(Input := "DI1_0", DI := "PLC_Signals_DB".DI_1_0, TON_Timer := "DI_1_0_TON", TOF_Timer := "DI_1_0_TOF")
   END_RUNG
   // the same network as SCL:
   "DI"(Input := "DI1_0", DI := "PLC_Signals_DB".DI_1_0, TON_Timer := "DI_1_0_TON", TOF_Timer := "DI_1_0_TOF");
END_REGION

REGION Network 18: DI_1_1 Сигнализатор уровня max
   RUNG wire#powerrail
      "DI"(Input := "DI1_1", DI := "PLC_Signals_DB".DI_1_1, TON_Timer := "DI_1_1_TON", TOF_Timer := "DI_1_1_TOF")
   END_RUNG
   // the same network as SCL:
   "DI"(Input := "DI1_1", DI := "PLC_Signals_DB".DI_1_1, TON_Timer := "DI_1_1_TON", TOF_Timer := "DI_1_1_TOF");
END_REGION

REGION Network 19: DI_1_2 Клапан 1
   RUNG wire#powerrail
      "DI"(Input := "DI1_2", DI := "PLC_Signals_DB".DI_1_2, TON_Timer := "DI_1_2_TON", TOF_Timer := "DI_1_2_TOF")
   END_RUNG
   // the same network as SCL:
   "DI"(Input := "DI1_2", DI := "PLC_Signals_DB".DI_1_2, TON_Timer := "DI_1_2_TON", TOF_Timer := "DI_1_2_TOF");
END_REGION

REGION Network 20: DI_1_3 Клапан 2
   RUNG wire#powerrail
      "DI"(Input := "DI1_3", DI := "PLC_Signals_DB".DI_1_3, TON_Timer := "DI_1_3_TON", TOF_Timer := "DI_1_3_TOF")
   END_RUNG
   // the same network as SCL:
   "DI"(Input := "DI1_3", DI := "PLC_Signals_DB".DI_1_3, TON_Timer := "DI_1_3_TON", TOF_Timer := "DI_1_3_TOF");
END_REGION

REGION Network 21: DI_1_4 Резерв
   RUNG wire#powerrail
      "DI"(Input := "DI1_4", DI := "PLC_Signals_DB".DI_1_4, TON_Timer := "DI_1_4_TON", TOF_Timer := "DI_1_4_TOF")
   END_RUNG
   // the same network as SCL:
   "DI"(Input := "DI1_4", DI := "PLC_Signals_DB".DI_1_4, TON_Timer := "DI_1_4_TON", TOF_Timer := "DI_1_4_TOF");
END_REGION

REGION Network 22: DI_1_5 Резерв
   RUNG wire#powerrail
      "DI"(Input := "DI1_5", DI := "PLC_Signals_DB".DI_1_5, TON_Timer := "DI_1_5_TON", TOF_Timer := "DI_1_5_TOF")
   END_RUNG
   // the same network as SCL:
   "DI"(Input := "DI1_5", DI := "PLC_Signals_DB".DI_1_5, TON_Timer := "DI_1_5_TON", TOF_Timer := "DI_1_5_TOF");
END_REGION

REGION Network 23: DI_1_6 Работа горелки
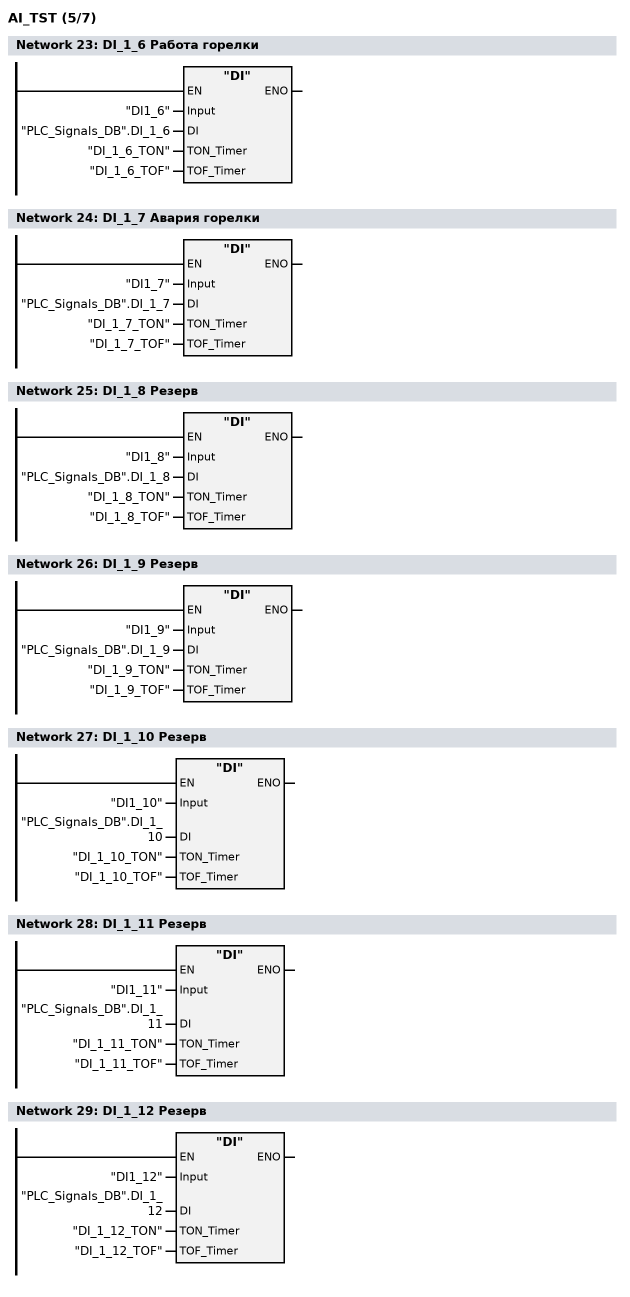
   RUNG wire#powerrail
      "DI"(Input := "DI1_6", DI := "PLC_Signals_DB".DI_1_6, TON_Timer := "DI_1_6_TON", TOF_Timer := "DI_1_6_TOF")
   END_RUNG
   // the same network as SCL:
   "DI"(Input := "DI1_6", DI := "PLC_Signals_DB".DI_1_6, TON_Timer := "DI_1_6_TON", TOF_Timer := "DI_1_6_TOF");
END_REGION

REGION Network 24: DI_1_7 Авария горелки
   RUNG wire#powerrail
      "DI"(Input := "DI1_7", DI := "PLC_Signals_DB".DI_1_7, TON_Timer := "DI_1_7_TON", TOF_Timer := "DI_1_7_TOF")
   END_RUNG
   // the same network as SCL:
   "DI"(Input := "DI1_7", DI := "PLC_Signals_DB".DI_1_7, TON_Timer := "DI_1_7_TON", TOF_Timer := "DI_1_7_TOF");
END_REGION

REGION Network 25: DI_1_8 Резерв
   RUNG wire#powerrail
      "DI"(Input := "DI1_8", DI := "PLC_Signals_DB".DI_1_8, TON_Timer := "DI_1_8_TON", TOF_Timer := "DI_1_8_TOF")
   END_RUNG
   // the same network as SCL:
   "DI"(Input := "DI1_8", DI := "PLC_Signals_DB".DI_1_8, TON_Timer := "DI_1_8_TON", TOF_Timer := "DI_1_8_TOF");
END_REGION

REGION Network 26: DI_1_9 Резерв
   RUNG wire#powerrail
      "DI"(Input := "DI1_9", DI := "PLC_Signals_DB".DI_1_9, TON_Timer := "DI_1_9_TON", TOF_Timer := "DI_1_9_TOF")
   END_RUNG
   // the same network as SCL:
   "DI"(Input := "DI1_9", DI := "PLC_Signals_DB".DI_1_9, TON_Timer := "DI_1_9_TON", TOF_Timer := "DI_1_9_TOF");
END_REGION

REGION Network 27: DI_1_10 Резерв
   RUNG wire#powerrail
      "DI"(Input := "DI1_10", DI := "PLC_Signals_DB".DI_1_10, TON_Timer := "DI_1_10_TON", TOF_Timer := "DI_1_10_TOF")
   END_RUNG
   // the same network as SCL:
   "DI"(Input := "DI1_10",
        DI := "PLC_Signals_DB".DI_1_10,
        TON_Timer := "DI_1_10_TON",
        TOF_Timer := "DI_1_10_TOF");
END_REGION

REGION Network 28: DI_1_11 Резерв
   RUNG wire#powerrail
      "DI"(Input := "DI1_11", DI := "PLC_Signals_DB".DI_1_11, TON_Timer := "DI_1_11_TON", TOF_Timer := "DI_1_11_TOF")
   END_RUNG
   // the same network as SCL:
   "DI"(Input := "DI1_11",
        DI := "PLC_Signals_DB".DI_1_11,
        TON_Timer := "DI_1_11_TON",
        TOF_Timer := "DI_1_11_TOF");
END_REGION

REGION Network 29: DI_1_12 Резерв
   RUNG wire#powerrail
      "DI"(Input := "DI1_12", DI := "PLC_Signals_DB".DI_1_12, TON_Timer := "DI_1_12_TON", TOF_Timer := "DI_1_12_TOF")
   END_RUNG
   // the same network as SCL:
   "DI"(Input := "DI1_12",
        DI := "PLC_Signals_DB".DI_1_12,
        TON_Timer := "DI_1_12_TON",
        TOF_Timer := "DI_1_12_TOF");
END_REGION

REGION Network 30: DI_1_13 Резерв
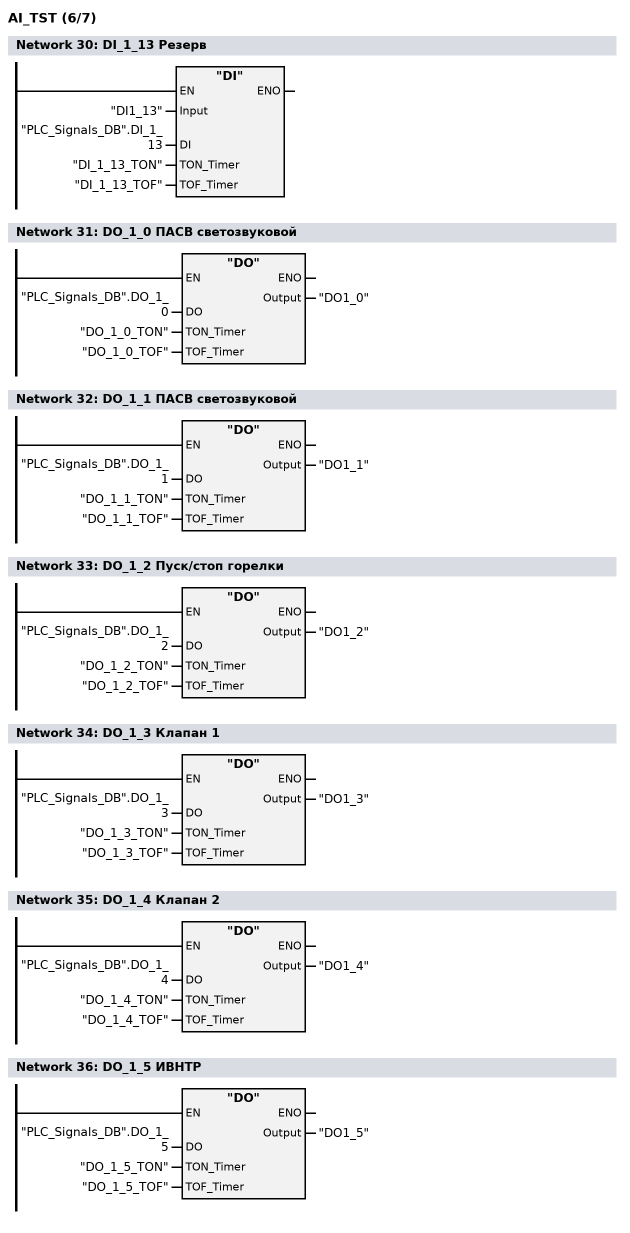
   RUNG wire#powerrail
      "DI"(Input := "DI1_13", DI := "PLC_Signals_DB".DI_1_13, TON_Timer := "DI_1_13_TON", TOF_Timer := "DI_1_13_TOF")
   END_RUNG
   // the same network as SCL:
   "DI"(Input := "DI1_13",
        DI := "PLC_Signals_DB".DI_1_13,
        TON_Timer := "DI_1_13_TON",
        TOF_Timer := "DI_1_13_TOF");
END_REGION

REGION Network 31: DO_1_0 ПАСВ светозвуковой
   RUNG wire#powerrail
      "DO"("DO" := "PLC_Signals_DB".DO_1_0, TON_Timer := "DO_1_0_TON", TOF_Timer := "DO_1_0_TOF", Output => "DO1_0")
   END_RUNG
   // the same network as SCL:
   "DO"("DO" := "PLC_Signals_DB".DO_1_0,
        TON_Timer := "DO_1_0_TON",
        TOF_Timer := "DO_1_0_TOF",
        Output => "DO1_0");
END_REGION

REGION Network 32: DO_1_1 ПАСВ светозвуковой
   RUNG wire#powerrail
      "DO"("DO" := "PLC_Signals_DB".DO_1_1, TON_Timer := "DO_1_1_TON", TOF_Timer := "DO_1_1_TOF", Output => "DO1_1")
   END_RUNG
   // the same network as SCL:
   "DO"("DO" := "PLC_Signals_DB".DO_1_1,
        TON_Timer := "DO_1_1_TON",
        TOF_Timer := "DO_1_1_TOF",
        Output => "DO1_1");
END_REGION

REGION Network 33: DO_1_2 Пуск/стоп горелки
   RUNG wire#powerrail
      "DO"("DO" := "PLC_Signals_DB".DO_1_2, TON_Timer := "DO_1_2_TON", TOF_Timer := "DO_1_2_TOF", Output => "DO1_2")
   END_RUNG
   // the same network as SCL:
   "DO"("DO" := "PLC_Signals_DB".DO_1_2,
        TON_Timer := "DO_1_2_TON",
        TOF_Timer := "DO_1_2_TOF",
        Output => "DO1_2");
END_REGION

REGION Network 34: DO_1_3 Клапан 1
   RUNG wire#powerrail
      "DO"("DO" := "PLC_Signals_DB".DO_1_3, TON_Timer := "DO_1_3_TON", TOF_Timer := "DO_1_3_TOF", Output => "DO1_3")
   END_RUNG
   // the same network as SCL:
   "DO"("DO" := "PLC_Signals_DB".DO_1_3,
        TON_Timer := "DO_1_3_TON",
        TOF_Timer := "DO_1_3_TOF",
        Output => "DO1_3");
END_REGION

REGION Network 35: DO_1_4 Клапан 2
   RUNG wire#powerrail
      "DO"("DO" := "PLC_Signals_DB".DO_1_4, TON_Timer := "DO_1_4_TON", TOF_Timer := "DO_1_4_TOF", Output => "DO1_4")
   END_RUNG
   // the same network as SCL:
   "DO"("DO" := "PLC_Signals_DB".DO_1_4,
        TON_Timer := "DO_1_4_TON",
        TOF_Timer := "DO_1_4_TOF",
        Output => "DO1_4");
END_REGION

REGION Network 36: DO_1_5 ИВНТР
   RUNG wire#powerrail
      "DO"("DO" := "PLC_Signals_DB".DO_1_5, TON_Timer := "DO_1_5_TON", TOF_Timer := "DO_1_5_TOF", Output => "DO1_5")
   END_RUNG
   // the same network as SCL:
   "DO"("DO" := "PLC_Signals_DB".DO_1_5,
        TON_Timer := "DO_1_5_TON",
        TOF_Timer := "DO_1_5_TOF",
        Output => "DO1_5");
END_REGION

REGION Network 37: DO_1_6 Резерв
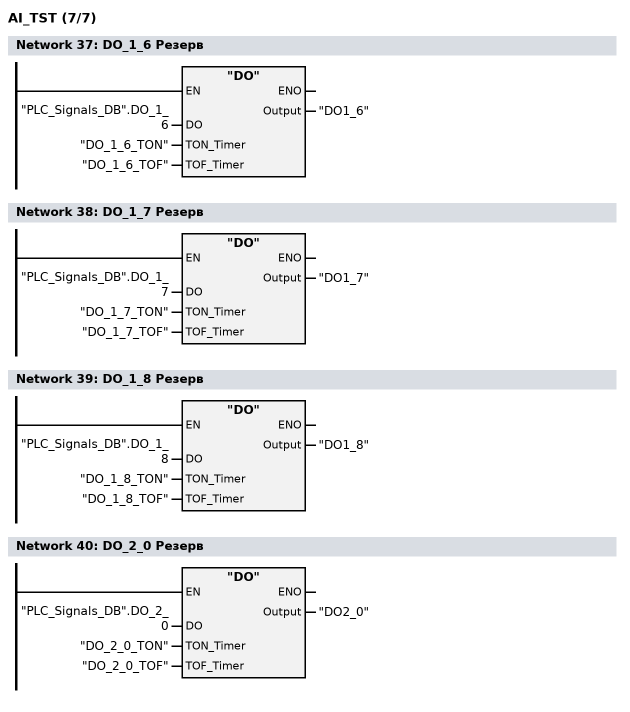
   RUNG wire#powerrail
      "DO"("DO" := "PLC_Signals_DB".DO_1_6, TON_Timer := "DO_1_6_TON", TOF_Timer := "DO_1_6_TOF", Output => "DO1_6")
   END_RUNG
   // the same network as SCL:
   "DO"("DO" := "PLC_Signals_DB".DO_1_6,
        TON_Timer := "DO_1_6_TON",
        TOF_Timer := "DO_1_6_TOF",
        Output => "DO1_6");
END_REGION

REGION Network 38: DO_1_7 Резерв
   RUNG wire#powerrail
      "DO"("DO" := "PLC_Signals_DB".DO_1_7, TON_Timer := "DO_1_7_TON", TOF_Timer := "DO_1_7_TOF", Output => "DO1_7")
   END_RUNG
   // the same network as SCL:
   "DO"("DO" := "PLC_Signals_DB".DO_1_7,
        TON_Timer := "DO_1_7_TON",
        TOF_Timer := "DO_1_7_TOF",
        Output => "DO1_7");
END_REGION

REGION Network 39: DO_1_8 Резерв
   RUNG wire#powerrail
      "DO"("DO" := "PLC_Signals_DB".DO_1_8, TON_Timer := "DO_1_8_TON", TOF_Timer := "DO_1_8_TOF", Output => "DO1_8")
   END_RUNG
   // the same network as SCL:
   "DO"("DO" := "PLC_Signals_DB".DO_1_8,
        TON_Timer := "DO_1_8_TON",
        TOF_Timer := "DO_1_8_TOF",
        Output => "DO1_8");
END_REGION

REGION Network 40: DO_2_0 Резерв
   RUNG wire#powerrail
      "DO"("DO" := "PLC_Signals_DB".DO_2_0, TON_Timer := "DO_2_0_TON", TOF_Timer := "DO_2_0_TOF", Output => "DO2_0")
   END_RUNG
   // the same network as SCL:
   "DO"("DO" := "PLC_Signals_DB".DO_2_0,
        TON_Timer := "DO_2_0_TON",
        TOF_Timer := "DO_2_0_TOF",
        Output => "DO2_0");
END_REGION
END_FUNCTION

FUNCTION "Valve_ctrl_1_0" : Void   // FC8, SCL
{ S7_Optimized_Access := 'TRUE' }
VERSION : 0.1
   VAR_INPUT
      Valve_opening : Bool;
      Valve_closing : Bool;
      Valve_Pos : Struct   // Аналоговый датчик положения клапана
         Hihi_Value : Real;   // Уставка: Hihi
         High_Value : Real;   // Уставка: High
         Low_Value : Real;   // Уставка: Low
         Lolo_Value : Real;   // Уставка: Lolo
         MIN_Current : Real;   // Настройка: Минимальное входное значение тока
         MAX_Current : Real;   // Настройка: Максимальное входное значение тока
         MAX_Value : Real;   // Настройка: Максимальное значение измеряемой величины
         MIN_Value : Real;   // Настройка: Минимальное значение измеряемой величины
         Underflow_RAW : Real;   // Настройка: Значение кода ацп при обрыве
         Overflow_RAW : Real;   // Настройка: Значение кода ацп при зашкале
         SCALED : Real;   // Выход: Масштабированное в инженерные единицы значение входного сигнала
         ING_Value : Real;   // Выход: Токовое значение датчика
         Manual_Value : Real;   // Значение, введенное вручную
         Alarm_Delay : Int;   // Настройка: Задержка срабатывания аварий
         Warning_Delay : Int;   // Настройка: Задержка срабатывания предупреждений
         AVG_Delay : Real;   // Настройка: Зона нечувствительности
         Underflow_Delay : Int;   // Настройка: Задержка отображения обрыва датчика
         Overflow_Delay : Int;   // Настройка: Задержка отображения неисправности датчика
         State : Word;   // Выход: Состояние датчика
         Modeee : Word;   // Настройка: Режим работы датчика
         bools : Word;   // Все булевы параметры AI
         AI_RAW_MIN : Int;   // Мин кода ацп
         AI_RAW_MAX : Int;   // Макс кода ацп
         Hihi_EN : Bool;   // Разрешение на сработку
         High_EN : Bool;   // Разрешение на сработку
         Low_En : Bool;   // Разрешение на сработку
         Lolo_EN : Bool;   // Разрешение на сработку
      END_STRUCT;
      Press_Out : Struct   // Аналоговый датчик положения клапана
         Hihi_Value : Real;   // Уставка: Hihi
         High_Value : Real;   // Уставка: High
         Low_Value : Real;   // Уставка: Low
         Lolo_Value : Real;   // Уставка: Lolo
         MIN_Current : Real;   // Настройка: Минимальное входное значение тока
         MAX_Current : Real;   // Настройка: Максимальное входное значение тока
         MAX_Value : Real;   // Настройка: Максимальное значение измеряемой величины
         MIN_Value : Real;   // Настройка: Минимальное значение измеряемой величины
         Underflow_RAW : Real;   // Настройка: Значение кода ацп при обрыве
         Overflow_RAW : Real;   // Настройка: Значение кода ацп при зашкале
         SCALED : Real;   // Выход: Масштабированное в инженерные единицы значение входного сигнала
         ING_Value : Real;   // Выход: Токовое значение датчика
         Manual_Value : Real;   // Значение, введенное вручную
         Alarm_Delay : Int;   // Настройка: Задержка срабатывания аварий
         Warning_Delay : Int;   // Настройка: Задержка срабатывания предупреждений
         AVG_Delay : Real;   // Настройка: Зона нечувствительности
         Underflow_Delay : Int;   // Настройка: Задержка отображения обрыва датчика
         Overflow_Delay : Int;   // Настройка: Задержка отображения неисправности датчика
         State : Word;   // Выход: Состояние датчика
         Modeee : Word;   // Настройка: Режим работы датчика
         bools : Word;   // Все булевы параметры AI
         AI_RAW_MIN : Int;   // Мин кода ацп
         AI_RAW_MAX : Int;   // Макс кода ацп
         Hihi_EN : Bool;   // Разрешение на сработку
         High_EN : Bool;   // Разрешение на сработку
         Low_En : Bool;   // Разрешение на сработку
         Lolo_EN : Bool;   // Разрешение на сработку
      END_STRUCT;
      Max_Open : Real;   // Максимальное открытие регулятора
   END_VAR
   VAR_OUTPUT
      CMD_Open_Out : Bool;
      CMD_Close_Out : Bool;
   END_VAR
   VAR_IN_OUT
      valve : Struct
         CMD_Open : Bool;   // Команда открыть
         CMD_Close : Bool;   // Команда закрыть
         CMD_ALRM_Stop : Bool;
         State : Word;
         State_INT : Int;
         Mode : Bool;   // 0-ручной, 1-авто
         Alarm : Word;
         bools : Word;
         RST_ALRM : Bool;
         CMD_Open_Out : Bool;   // управление открыть
         CMD_Close_Out : Bool;   // управление закрыть
         Press_Need : Real;   // Уставка по давлению
         Press_Need_Open : Real;   // Разница между уставно и текущим давлением
         Press_Need_Close : Real;   // Разница между уставно и текущим давлением
         Press_Need_Open_Perc : Real;
         Press_Need_Close_Perc : Real;
      END_STRUCT;
      TIME_Opening : TON_TIME;
      TIME_Closing : TON_TIME;
   END_VAR
BEGIN
   IF #Valve_Pos.State.%X5 OR #Valve_Pos.State.%X6 THEN
       #valve.Alarm.%X0 := TRUE;
   END_IF;
   #valve.State.%X0 := #valve.Alarm.%X0;


   //ручной режим
   IF NOT (#valve.Mode) THEN

       IF #valve.Alarm = 0 THEN
           #valve.CMD_Open_Out := #valve.CMD_Open;
           #valve.CMD_Close_Out := #valve.CMD_Close;
       ELSE
           #valve.CMD_Open_Out := FALSE;
           #valve.CMD_Close_Out := FALSE;
       END_IF;

   END_IF;

   //автоматический режим
   (* IF #valve.Mode THEN

       #valve.Press_Need_Open := 

   END_IF; *)

   #valve.Press_Need_Open_Perc := (#valve.Press_Need * 5) / 100;
   #valve.Press_Need_Open := #valve.Press_Need - #valve.Press_Need_Open_Perc;
   #valve.Press_Need_Close_Perc := (#valve.Press_Need * 5) / 100;
   #valve.Press_Need_Close := #valve.Press_Need + #valve.Press_Need_Open_Perc;

   IF #valve.Mode THEN

       IF #Press_Out.SCALED < #valve.Press_Need_Open THEN
           #valve.CMD_Open_Out := TRUE;
       ELSE
           #valve.CMD_Open_Out := FALSE;
       END_IF;
       IF #Press_Out.SCALED > #valve.Press_Need_Close THEN
           #valve.CMD_Close_Out := TRUE;
       ELSE
           #valve.CMD_Close_Out := FALSE;
       END_IF;

       IF #valve.CMD_ALRM_Stop OR #valve.Alarm <> 0 THEN
           #valve.CMD_Open_Out := FALSE;
           #valve.CMD_Close_Out := FALSE;
       END_IF;
       IF #valve.CMD_Open OR #valve.CMD_Close THEN
           #valve.CMD_ALRM_Stop := 0;
       END_IF;

   END_IF;



   IF #Valve_Pos.SCALED >= 100(*#Valve_Pos.MAX_Value*)THEN
       //#valve.CMD_Open_Out := FALSE;
       #valve.State.%X5 := TRUE;
   ELSE
       #valve.State.%X5 := FALSE;
   END_IF;
   IF #Valve_Pos.SCALED <= 0 (*#Valve_Pos.MIN_Value*)THEN
       #valve.CMD_Close_Out := FALSE;
       #valve.State.%X6 := TRUE;
   ELSE
       #valve.State.%X6 := FALSE;
   END_IF;

   //формирование состояний
   #valve.State.%X3 := #Valve_opening;
   #valve.State.%X4 := #Valve_closing;
   IF NOT (#Valve_opening) AND NOT (#Valve_closing) THEN
       #valve.State.%X7 := TRUE;
   ELSE
       #valve.State.%X7 := FALSE;
   END_IF;

   IF #Valve_Pos.SCALED >= #Max_Open AND #valve.Mode THEN
       #valve.CMD_Open_Out := FALSE;
   END_IF;

   //аварии при открытии и закрытии
   #TIME_Opening.TON(IN := #valve.CMD_Open_Out AND NOT (#Valve_opening),
                     PT := T#5s);
   IF #TIME_Opening.Q THEN
       #valve.Alarm.%X1 := TRUE;
   END_IF;
   #valve.State.%X1 := #valve.Alarm.%X1;

   #TIME_Closing.TON(IN := #valve.CMD_Close_Out AND NOT (#Valve_closing),
                     PT := T#5s);
   IF #TIME_Closing.Q THEN
       #valve.Alarm.%X2 := TRUE;
   END_IF;
   #valve.State.%X2 := #valve.Alarm.%X2;




   //Состояниея в Int
   IF #valve.State.%X0 THEN
       #valve.State_INT := 0;
   ELSIF #valve.State.%X1 THEN
       #valve.State_INT := 1;
   ELSIF #valve.State.%X2 THEN
       #valve.State_INT := 2;
   ELSIF #valve.State.%X3 THEN
       #valve.State_INT := 3;
   ELSIF #valve.State.%X4 THEN
       #valve.State_INT := 4;
   ELSIF #valve.State.%X5 THEN
       #valve.State_INT := 5;
   ELSIF #valve.State.%X6 THEN
       #valve.State_INT := 6;
   ELSIF #valve.State.%X7 THEN
       #valve.State_INT := 7;
   END_IF;



   IF #valve.RST_ALRM THEN
       #valve.Alarm := 0;
   END_IF;

   #CMD_Open_Out := #valve.CMD_Open_Out;
   #CMD_Close_Out := #valve.CMD_Close_Out;
END_FUNCTION

FUNCTION "Vent" : Void   // FC9, LAD
{ S7_Optimized_Access := 'TRUE' }
VERSION : 0.1
   VAR_INPUT
      QT_State : Int;
      Vent_State : Bool;
      Dostup : Bool;
      Fire : Bool;
      Avar_stop : Bool;
   END_VAR
   VAR_OUTPUT
      Pusk : Bool;
      Stop : Bool;
   END_VAR
   VAR_TEMP
      pt_time : Time;
      et_time : Time;
   END_VAR
BEGIN

REGION Network 1
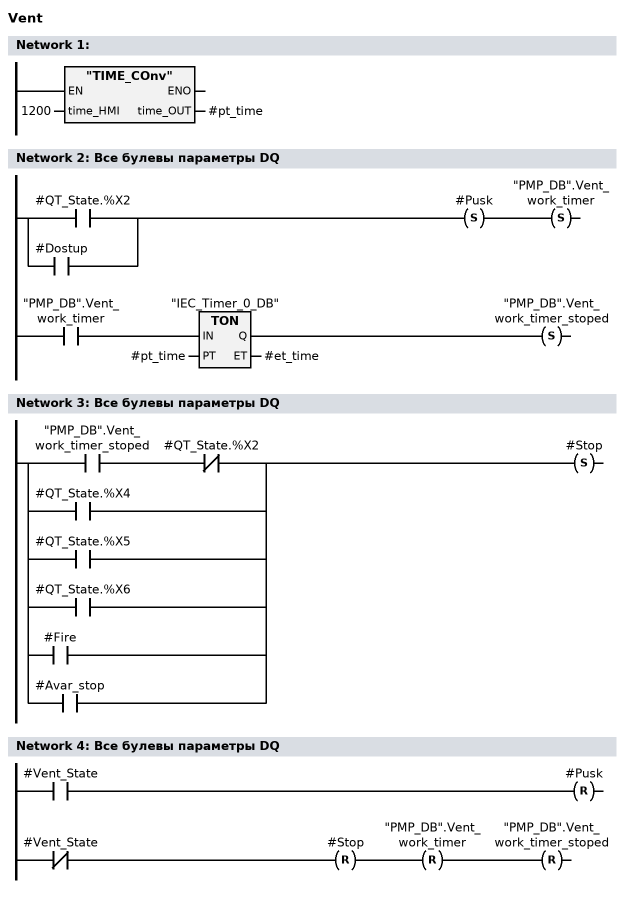
   RUNG wire#powerrail
      "TIME_COnv"(time_HMI := 1200, time_OUT => #pt_time)
   END_RUNG
   // the same network as SCL:
   "TIME_COnv"(time_HMI := 1200, time_OUT => #pt_time);
END_REGION

REGION Network 2: Все булевы параметры DQ
   IF #QT_State.%X2 OR #Dostup THEN
       #Pusk := TRUE;
       "PMP_DB".Vent_work_timer := TRUE;
   END_IF;
   "IEC_Timer_0_DB".TON(IN := "PMP_DB".Vent_work_timer, PT := #pt_time, ET => #et_time);
   IF "IEC_Timer_0_DB".Q THEN "PMP_DB".Vent_work_timer_stoped := TRUE; END_IF;
END_REGION

REGION Network 3: Все булевы параметры DQ
   RUNG wire#powerrail
      Contact( "PMP_DB".Vent_work_timer_stoped )
      I_Contact( #QT_State.%X2 )
      wire#w1
      S_Coil( #Stop )
   END_RUNG
   RUNG wire#powerrail
      Contact( #QT_State.%X4 )
   END_RUNG wire#w1
   RUNG wire#powerrail
      Contact( #QT_State.%X5 )
   END_RUNG wire#w1
   RUNG wire#powerrail
      Contact( #QT_State.%X6 )
   END_RUNG wire#w1
   RUNG wire#powerrail
      Contact( #Fire )
   END_RUNG wire#w1
   RUNG wire#powerrail
      Contact( #Avar_stop )
   END_RUNG wire#w1
   // the same network as SCL:
   IF ("PMP_DB".Vent_work_timer_stoped AND NOT #QT_State.%X2) OR #QT_State.%X4 OR #QT_State.%X5 OR #QT_State.%X6 OR #Fire OR #Avar_stop THEN
       #Stop := TRUE;
   END_IF;
END_REGION

REGION Network 4: Все булевы параметры DQ
   RUNG wire#powerrail
      Contact( #Vent_State )
      R_Coil( #Pusk )
   END_RUNG
   RUNG wire#powerrail
      I_Contact( #Vent_State )
      R_Coil( #Stop )
      R_Coil( "PMP_DB".Vent_work_timer )
      R_Coil( "PMP_DB".Vent_work_timer_stoped )
   END_RUNG
   // the same network as SCL:
   IF #Vent_State THEN #Pusk := FALSE; END_IF;
   IF NOT #Vent_State THEN
       #Stop := FALSE;
       "PMP_DB".Vent_work_timer := FALSE;
       "PMP_DB".Vent_work_timer_stoped := FALSE;
   END_IF;
END_REGION
END_FUNCTION

FUNCTION "MB_SLave_Transmision" : Void   // FC10, SCL
{ S7_Optimized_Access := 'TRUE' }
VERSION : 0.1
BEGIN
   (*"Slave".MBVerh_0 :=  REAL_TO_INT ("PLC_Signals_DB".AI_2_0.SCALED * 100);
   "Slave".MBVerh_1 :=  REAL_TO_INT ("PLC_Signals_DB".AI_2_1.SCALED * 100);
   "Slave".MBVerh_2 :=  REAL_TO_INT ("PLC_Signals_DB".AI_2_2.SCALED * 100);
   "Slave".MBVerh_3 :=  REAL_TO_INT ("PLC_Signals_DB".AI_2_3.SCALED * 100);
   "Slave".MBVerh_4 :=  REAL_TO_INT ("PLC_Signals_DB".AI_2_4.SCALED * 100);
   "Slave".MBVerh_5 :=  REAL_TO_INT ("PLC_Signals_DB".AI_2_5.SCALED * 100);
   "Slave".MBVerh_6 :=  REAL_TO_INT ("PLC_Signals_DB".AI_2_6.SCALED * 100);

   "Slave".MBVerh_7.%X0 := "PLC_Signals_DB".DI_1_0.Output;
   "Slave".MBVerh_7.%X1 := "PLC_Signals_DB".DI_1_1.Output;
   "Slave".MBVerh_7.%X2 := "PLC_Signals_DB".DI_1_2.Output;
   "Slave".MBVerh_7.%X3 := "PLC_Signals_DB".DI_1_3.Output;
   "Slave".MBVerh_7.%X4 := "PLC_Signals_DB".DI_1_6.Output;
   "Slave".MBVerh_7.%X5 := "PLC_Signals_DB".DI_1_7.Output;
   "Slave".MBVerh_7.%X6 := "PLC_Signals_DB".AI_2_6.State.%X2;
   "Slave".MBVerh_7.%X7 := "PLC_Signals_DB".AI_2_6.State.%X1;
   "Slave".MBVerh_7.%X8 := "PLC_Signals_DB".AI_2_6.State.%X5;
   "Slave".MBVerh_7.%X9 := "DB_TST".Valve_alarm_1;
   "Slave".MBVerh_7.%X10 := "DB_TST".Valve_alarm_2;


   "Slave".MBVerh_8.%X0 := "PLC_Signals_DB".AI_2_0.State.%X1;
   "Slave".MBVerh_8.%X1 := "PLC_Signals_DB".AI_2_1.State.%X1;
   "Slave".MBVerh_8.%X2 := "PLC_Signals_DB".AI_2_2.State.%X1;
   "Slave".MBVerh_8.%X3 := "PLC_Signals_DB".AI_2_3.State.%X1;
   "Slave".MBVerh_8.%X4 := "PLC_Signals_DB".AI_2_4.State.%X1;
   "Slave".MBVerh_8.%X5 := "PLC_Signals_DB".AI_2_5.State.%X1;
   "Slave".MBVerh_8.%X6 := "PLC_Signals_DB".AI_2_6.State.%X1;
   "Slave".MBVerh_8.%X7 := "PLC_Signals_DB".AI_2_0.State.%X2;
   "Slave".MBVerh_8.%X8 := "PLC_Signals_DB".AI_2_1.State.%X2;
   "Slave".MBVerh_8.%X9 := "PLC_Signals_DB".AI_2_2.State.%X2;
   "Slave".MBVerh_8.%X10 := "PLC_Signals_DB".AI_2_3.State.%X2;
   "Slave".MBVerh_8.%X11 := "PLC_Signals_DB".AI_2_4.State.%X2;
   "Slave".MBVerh_8.%X12 := "PLC_Signals_DB".AI_2_5.State.%X2;
   "Slave".MBVerh_8.%X13 := "PLC_Signals_DB".AI_2_6.State.%X2;


   "Slave".MBVerh_9.%X0 := "PLC_Signals_DB".AI_2_0.State.%X3;
   "Slave".MBVerh_9.%X1 := "PLC_Signals_DB".AI_2_1.State.%X3;
   "Slave".MBVerh_9.%X2 := "PLC_Signals_DB".AI_2_2.State.%X3;
   "Slave".MBVerh_9.%X3 := "PLC_Signals_DB".AI_2_3.State.%X3;
   "Slave".MBVerh_9.%X4 := "PLC_Signals_DB".AI_2_4.State.%X3;
   "Slave".MBVerh_9.%X5 := "PLC_Signals_DB".AI_2_5.State.%X3;
   "Slave".MBVerh_9.%X6 := "PLC_Signals_DB".AI_2_6.State.%X3;
   "Slave".MBVerh_9.%X7 := "PLC_Signals_DB".AI_2_0.State.%X4;
   "Slave".MBVerh_9.%X8 := "PLC_Signals_DB".AI_2_1.State.%X4;
   "Slave".MBVerh_9.%X9 := "PLC_Signals_DB".AI_2_2.State.%X4;
   "Slave".MBVerh_9.%X10 := "PLC_Signals_DB".AI_2_3.State.%X4;
   "Slave".MBVerh_9.%X11 := "PLC_Signals_DB".AI_2_4.State.%X4;
   "Slave".MBVerh_9.%X12 := "PLC_Signals_DB".AI_2_5.State.%X4;
   "Slave".MBVerh_9.%X13 := "PLC_Signals_DB".AI_2_6.State.%X4;


   "Slave".MBVerh_10.%X0 := "DB_TST".Burner.State = 0;
   "Slave".MBVerh_10.%X1 := "DB_TST".Burner.State = 1;
   "Slave".MBVerh_10.%X2 := "DB_TST".Burner.State = 2;
   "Slave".MBVerh_10.%X3 := NOT "DB_TST".Burner.mode;
   "Slave".MBVerh_10.%X4 := "DB_TST".Burner.mode;


   "Slave".MBVerh_11 := REAL_TO_INT (("DB_TST".T_Emk_Lo_Hmi) * 100);
   "Slave".MBVerh_12 := REAL_TO_INT (("DB_TST".T_Emk_Hi_Hmi) * 100);
   "Slave".MBVerh_13 := REAL_TO_INT (("DB_TST".T_Oil_Lo_Hmi) * 100);
   "Slave".MBVerh_14 := REAL_TO_INT (("DB_TST".T_Oil_Hi_Hmi) * 100);

   "DB_TST".Burner.ARM_start := "Slave".MBVerh_15.%X0;
   "DB_TST".Burner.ARM_stop := "Slave".MBVerh_15.%X1;
   "DB_TST".Burner.ARM_deblock := "Slave".MBVerh_15.%X2;
   "DB_TST".Burner.mode_ARM := "Slave".MBVerh_15.%X3;


   "DB_TST".P_gaz_out.Hihi := "PLC_Signals_DB".AI_2_0.State.%X1;
   "DB_TST".P_gaz_out.Hi := "PLC_Signals_DB".AI_2_0.State.%X2;
   "DB_TST".P_gaz_out.Lo := "PLC_Signals_DB".AI_2_0.State.%X3;
   "DB_TST".P_gaz_out.Lolo := "PLC_Signals_DB".AI_2_0.State.%X4;

   "DB_TST".P_gaz_in.Hihi := "PLC_Signals_DB".AI_2_1.State.%X1;
   "DB_TST".P_gaz_in.Hi := "PLC_Signals_DB".AI_2_1.State.%X2;
   "DB_TST".P_gaz_in.Lo := "PLC_Signals_DB".AI_2_1.State.%X3;
   "DB_TST".P_gaz_in.Lolo := "PLC_Signals_DB".AI_2_1.State.%X4;

   "DB_TST".P_gaza.Hihi := "PLC_Signals_DB".AI_2_2.State.%X1;
   "DB_TST".P_gaza.Hi := "PLC_Signals_DB".AI_2_2.State.%X2;
   "DB_TST".P_gaza.Lo := "PLC_Signals_DB".AI_2_2.State.%X3;
   "DB_TST".P_gaza.Lolo := "PLC_Signals_DB".AI_2_2.State.%X4;

   "DB_TST".T_gaza_out.Hihi := "PLC_Signals_DB".AI_2_3.State.%X1;
   "DB_TST".T_gaza_out.Hi := "PLC_Signals_DB".AI_2_3.State.%X2;
   "DB_TST".T_gaza_out.Lo := "PLC_Signals_DB".AI_2_3.State.%X3;
   "DB_TST".T_gaza_out.Lolo := "PLC_Signals_DB".AI_2_3.State.%X4;

   "DB_TST".T_dym_gazov.Hihi := "PLC_Signals_DB".AI_2_4.State.%X1;
   "DB_TST".T_dym_gazov.Hi := "PLC_Signals_DB".AI_2_4.State.%X2;
   "DB_TST".T_dym_gazov.Lo := "PLC_Signals_DB".AI_2_4.State.%X3;
   "DB_TST".T_dym_gazov.Lolo := "PLC_Signals_DB".AI_2_4.State.%X4;

   "DB_TST".T_emk.Hihi := "PLC_Signals_DB".AI_2_5.State.%X1;
   "DB_TST".T_emk.Hi := "PLC_Signals_DB".AI_2_5.State.%X2;
   "DB_TST".T_emk.Lo := "PLC_Signals_DB".AI_2_5.State.%X3;
   "DB_TST".T_emk.Lolo := "PLC_Signals_DB".AI_2_5.State.%X4;

   "DB_TST".Gazik.Hihi := "PLC_Signals_DB".AI_2_6.State.%X1;
   "DB_TST".Gazik.Hi := "PLC_Signals_DB".AI_2_6.State.%X2;
   "DB_TST".Gazik.Lo := "PLC_Signals_DB".AI_2_6.State.%X3;
   "DB_TST".Gazik.Lolo := "PLC_Signals_DB".AI_2_6.State.%X4;

   //Режим горелки
   IF "DB_TST".Burner.mode_ARM OR "DB_TST".Burner.mode_Hmi THEN
       "DB_TST".Burner.mode := 1;
   ELSE
       "DB_TST".Burner.mode := 0;
   END_IF;*)

   "Slave".MBVerh_0 := REAL_TO_INT("PLC_Signals_DB".AI_2_0.SCALED * 100);
   "Slave".MBVerh_1 := REAL_TO_INT("PLC_Signals_DB".AI_2_1.SCALED * 100);
   "Slave".MBVerh_2 := REAL_TO_INT("PLC_Signals_DB".AI_2_2.SCALED * 100);
   "Slave".MBVerh_3 := REAL_TO_INT("PLC_Signals_DB".AI_2_3.SCALED * 100);
   "Slave".MBVerh_4 := REAL_TO_INT("PLC_Signals_DB".AI_2_4.SCALED * 100);
   "Slave".MBVerh_5 := REAL_TO_INT("PLC_Signals_DB".AI_2_5.SCALED * 100);
   "Slave".MBVerh_6 := REAL_TO_INT("PLC_Signals_DB".AI_2_6.SCALED * 100);
   "Slave".MBVerh_7 := REAL_TO_INT("PLC_Signals_DB".AI_2_7.SCALED);

   "Slave".MBVerh_8.%X0 := "PLC_Signals_DB".DI_1_0.Output;
   "Slave".MBVerh_8.%X1 := "PLC_Signals_DB".DI_1_1.Output;
   "Slave".MBVerh_8.%X2 := "PLC_Signals_DB".DI_1_2.Output;
   "Slave".MBVerh_8.%X3 := "PLC_Signals_DB".DI_1_3.Output;
   "Slave".MBVerh_8.%X4 := "PLC_Signals_DB".DI_1_6.Output;
   "Slave".MBVerh_8.%X5 := "PLC_Signals_DB".DI_1_7.Output;
   "Slave".MBVerh_8.%X6 := "PLC_Signals_DB".AI_2_6.State.%X2;
   "Slave".MBVerh_8.%X7 := "PLC_Signals_DB".AI_2_6.State.%X1;
   "Slave".MBVerh_8.%X8 := "PLC_Signals_DB".AI_2_6.State.%X5;
   "Slave".MBVerh_8.%X9 := "DB_TST".Valve_alarm_1;
   "Slave".MBVerh_8.%X10 := "DB_TST".Valve_alarm_2;

   "Slave".MBVerh_9.%X0 := "PLC_Signals_DB".AI_2_0.State.%X1;
   "Slave".MBVerh_9.%X1 := "PLC_Signals_DB".AI_2_1.State.%X1;
   "Slave".MBVerh_9.%X2 := "PLC_Signals_DB".AI_2_2.State.%X1;
   "Slave".MBVerh_9.%X3 := "PLC_Signals_DB".AI_2_3.State.%X1;
   "Slave".MBVerh_9.%X4 := "PLC_Signals_DB".AI_2_4.State.%X1;
   "Slave".MBVerh_9.%X5 := "PLC_Signals_DB".AI_2_5.State.%X1;
   "Slave".MBVerh_9.%X6 := "PLC_Signals_DB".AI_2_6.State.%X1;
   "Slave".MBVerh_9.%X7 := "PLC_Signals_DB".AI_2_7.State.%X1;
   "Slave".MBVerh_9.%X8 := "PLC_Signals_DB".AI_2_0.State.%X2;
   "Slave".MBVerh_9.%X9 := "PLC_Signals_DB".AI_2_1.State.%X2;
   "Slave".MBVerh_9.%X10 := "PLC_Signals_DB".AI_2_2.State.%X2;
   "Slave".MBVerh_9.%X11 := "PLC_Signals_DB".AI_2_3.State.%X2;
   "Slave".MBVerh_9.%X12 := "PLC_Signals_DB".AI_2_4.State.%X2;
   "Slave".MBVerh_9.%X13 := "PLC_Signals_DB".AI_2_5.State.%X2;
   "Slave".MBVerh_9.%X14 := "PLC_Signals_DB".AI_2_6.State.%X2;
   "Slave".MBVerh_9.%X15 := "PLC_Signals_DB".AI_2_7.State.%X2;

   "Slave".MBVerh_10.%X0 := "PLC_Signals_DB".AI_2_0.State.%X3;
   "Slave".MBVerh_10.%X1 := "PLC_Signals_DB".AI_2_1.State.%X3;
   "Slave".MBVerh_10.%X2 := "PLC_Signals_DB".AI_2_2.State.%X3;
   "Slave".MBVerh_10.%X3 := "PLC_Signals_DB".AI_2_3.State.%X3;
   "Slave".MBVerh_10.%X4 := "PLC_Signals_DB".AI_2_4.State.%X3;
   "Slave".MBVerh_10.%X5 := "PLC_Signals_DB".AI_2_5.State.%X3;
   "Slave".MBVerh_10.%X6 := "PLC_Signals_DB".AI_2_6.State.%X3;
   "Slave".MBVerh_10.%X7 := "PLC_Signals_DB".AI_2_7.State.%X3;
   "Slave".MBVerh_10.%X8 := "PLC_Signals_DB".AI_2_0.State.%X4;
   "Slave".MBVerh_10.%X9 := "PLC_Signals_DB".AI_2_1.State.%X4;
   "Slave".MBVerh_10.%X10 := "PLC_Signals_DB".AI_2_2.State.%X4;
   "Slave".MBVerh_10.%X11 := "PLC_Signals_DB".AI_2_3.State.%X4;
   "Slave".MBVerh_10.%X12 := "PLC_Signals_DB".AI_2_4.State.%X4;
   "Slave".MBVerh_10.%X13 := "PLC_Signals_DB".AI_2_5.State.%X4;
   "Slave".MBVerh_10.%X14 := "PLC_Signals_DB".AI_2_6.State.%X4;
   "Slave".MBVerh_10.%X15 := "PLC_Signals_DB".AI_2_7.State.%X4;

   "Slave".MBVerh_11.%X0 := "DB_TST".Burner.State = 0;
   "Slave".MBVerh_11.%X1 := "DB_TST".Burner.State = 1;
   "Slave".MBVerh_11.%X2 := "DB_TST".Burner.State = 2;
   "Slave".MBVerh_11.%X3 := NOT "DB_TST".Burner.mode;
   "Slave".MBVerh_11.%X4 := "DB_TST".Burner.mode;

   "Slave".MBVerh_12 := REAL_TO_INT(("DB_TST".T_Emk_Lo_Hmi) * 100);
   "Slave".MBVerh_13 := REAL_TO_INT(("DB_TST".T_Emk_Hi_Hmi) * 100);
   "Slave".MBVerh_14 := REAL_TO_INT(("DB_TST".T_Oil_Lo_Hmi) * 100);
   "Slave".MBVerh_15 := REAL_TO_INT(("DB_TST".T_Oil_Hi_Hmi) * 100);

   "DB_TST".Burner.ARM_start := "Slave".MBVerh_16.%X0;
   "DB_TST".Burner.ARM_stop := "Slave".MBVerh_16.%X1;
   "DB_TST".Burner.ARM_deblock := "Slave".MBVerh_16.%X2;
   "DB_TST".Burner.mode_ARM := "Slave".MBVerh_16.%X3;
   "DB_TST".Valve_1.RST_ALRM := "Slave".MBVerh_16.%X4;
   "DB_TST".Valve_2.RST_ALRM := "Slave".MBVerh_16.%X4;

   "DB_TST".P_gaz_out.Hihi := "PLC_Signals_DB".AI_2_0.State.%X1;
   "DB_TST".P_gaz_out.Hi := "PLC_Signals_DB".AI_2_0.State.%X2;
   "DB_TST".P_gaz_out.Lo := "PLC_Signals_DB".AI_2_0.State.%X3;
   "DB_TST".P_gaz_out.Lolo := "PLC_Signals_DB".AI_2_0.State.%X4;

   "DB_TST".P_gaz_in.Hihi := "PLC_Signals_DB".AI_2_1.State.%X1;
   "DB_TST".P_gaz_in.Hi := "PLC_Signals_DB".AI_2_1.State.%X2;
   "DB_TST".P_gaz_in.Lo := "PLC_Signals_DB".AI_2_1.State.%X3;
   "DB_TST".P_gaz_in.Lolo := "PLC_Signals_DB".AI_2_1.State.%X4;

   "DB_TST".P_gaza.Hihi := "PLC_Signals_DB".AI_2_2.State.%X1;
   "DB_TST".P_gaza.Hi := "PLC_Signals_DB".AI_2_2.State.%X2;
   "DB_TST".P_gaza.Lo := "PLC_Signals_DB".AI_2_2.State.%X3;
   "DB_TST".P_gaza.Lolo := "PLC_Signals_DB".AI_2_2.State.%X4;

   "DB_TST".T_gaza_out.Hihi := "PLC_Signals_DB".AI_2_3.State.%X1;
   "DB_TST".T_gaza_out.Hi := "PLC_Signals_DB".AI_2_3.State.%X2;
   "DB_TST".T_gaza_out.Lo := "PLC_Signals_DB".AI_2_3.State.%X3;
   "DB_TST".T_gaza_out.Lolo := "PLC_Signals_DB".AI_2_3.State.%X4;

   "DB_TST".T_dym_gazov.Hihi := "PLC_Signals_DB".AI_2_4.State.%X1;
   "DB_TST".T_dym_gazov.Hi := "PLC_Signals_DB".AI_2_4.State.%X2;
   "DB_TST".T_dym_gazov.Lo := "PLC_Signals_DB".AI_2_4.State.%X3;
   "DB_TST".T_dym_gazov.Lolo := "PLC_Signals_DB".AI_2_4.State.%X4;

   "DB_TST".T_emk.Hihi := "PLC_Signals_DB".AI_2_5.State.%X1;
   "DB_TST".T_emk.Hi := "PLC_Signals_DB".AI_2_5.State.%X2;
   "DB_TST".T_emk.Lo := "PLC_Signals_DB".AI_2_5.State.%X3;
   "DB_TST".T_emk.Lolo := "PLC_Signals_DB".AI_2_5.State.%X4;

   "DB_TST".T_emk_B1.Hihi := "PLC_Signals_DB".AI_2_6.State.%X1;
   "DB_TST".T_emk_B1.Hi := "PLC_Signals_DB".AI_2_6.State.%X2;
   "DB_TST".T_emk_B1.Lo := "PLC_Signals_DB".AI_2_6.State.%X3;
   "DB_TST".T_emk_B1.Lolo := "PLC_Signals_DB".AI_2_6.State.%X4;

   "DB_TST".Gazik.Hihi := "PLC_Signals_DB".AI_2_7.State.%X1;
   "DB_TST".Gazik.Hi := "PLC_Signals_DB".AI_2_7.State.%X2;
   "DB_TST".Gazik.Lo := "PLC_Signals_DB".AI_2_7.State.%X3;
   "DB_TST".Gazik.Lolo := "PLC_Signals_DB".AI_2_7.State.%X4;

   //Режим горелки
   IF "DB_TST".Burner.mode_ARM OR "DB_TST".Burner.mode_Hmi THEN
       "DB_TST".Burner.mode := 1;
   ELSE
       "DB_TST".Burner.mode := 0;
   END_IF;
END_FUNCTION

FUNCTION "Burner" : Void   // FC11, SCL
{ S7_Optimized_Access := 'TRUE' }
VERSION : 0.1
   VAR_INPUT
      Burn_Alarm : Bool;   // Авария горелки di
      Burn_Work : Bool;
      T_Gaz_HiHi : Bool;   // Аварийная уставка температуры дымовых газов max
      P_Gaz_HiHi_In : Bool;   // Аварийная уставка давление на входе max
      P_Gaz_LoLo_In : Bool;   // Аварийная уставка давление на входе min
      P_Gaz_HiHi_Out : Bool;   // Аварийная уставка давление на выходе max
      P_Gaz_LoLo_Out : Bool;   // Аварийная уставка давление на выходе min
      T_Emk_HiHi : Bool;   // Аварийная уставка температуры ёмкости max
      T_Oil_HiHi_Out : Bool;   // Аварийная уставка температуры на выходе max
      P_Gaz_LoLo : Bool;   // Аварийная уставка давление газа min
      P_Gaz_HiHi : Bool;   // Аварийная уставка давление газа max
      Porog_2 : Bool;   // Загазованность порог 2
      T_Emk : Real;
      T_Oil : Real;
      T_Need_Emk_Hi : Real;   // Максимальная температура в теплоносители
      T_Need_Oil_Hi : Real;   // Максимальная температура нефти
      T_Need_Emk_Lo : Real;
      T_Need_Oil_Lo : Real;
      Valve_alarm_1 : Bool;   // Аврия запальной горелки
      Valve_alarm_2 : Bool;   // Авария основной горелки
      State_open_cl_1 : Bool;   // Клапан на запальную горелку открыт
      H_HiHi : Bool;   // Аварийная уставка уровня max
      H_LoLo : Bool;   // Аварийная уставка уровня min
   END_VAR
   VAR_OUTPUT
      Burner_ON : Bool;
      RST_Block_Burner : Bool;
      Need_open_cl_1 : Bool;   // Открыть клапан на запальную горелку
      Need_open_cl_2 : Bool;   // Открыть клапан на основную горелку
      Burner_fire : Bool;   // Искра на горелку
   END_VAR
   VAR_IN_OUT
      Burner : Struct
         State_W : DWord;
         State : Int;
         CMD_Start : Bool;
         CMD_Stop : Bool;
         CMD_RST_Alarm : Bool;
         CMD_Start_Stop : Bool;
         Alarm_W : DWord;
         Alarm_INT : Int;
         Alarm : Bool;
         Auto_Pause : Bool;
         Flag_Auto_Pause : Bool;
         Fire : Bool;
         mode : Bool;   // 0-ручной/1-АРМ
         mode_Hmi : Bool;
         mode_ARM : Bool;
         ARM_start : Bool;
         ARM_stop : Bool;
         ARM_deblock : Bool;
      END_STRUCT;
      Timer_Not_Start : TON_TIME;
      Timer_need_cl_2 : TON_TIME;   // Задержка на открытие клапана на основную горелку
   END_VAR
BEGIN


   //формирование аварий
   (*IF #Burn_Alarm THEN
       #Burner.Alarm_W.%X1 := TRUE;
   END_IF;*)

   IF #T_Gaz_HiHi AND (#Burn_Work OR #Burner.CMD_Start OR #Burner.CMD_Start_Stop) THEN
       #Burner.Alarm_W.%X2 := TRUE;
   END_IF;

   IF #P_Gaz_LoLo_Out AND (#Burn_Work OR #Burner.CMD_Start OR #Burner.CMD_Start_Stop) THEN
       #Burner.Alarm_W.%X3 := TRUE;
   END_IF;

   IF #P_Gaz_HiHi_Out AND (#Burn_Work OR #Burner.CMD_Start OR #Burner.CMD_Start_Stop) THEN
       #Burner.Alarm_W.%X4 := TRUE;
   END_IF;

   IF #P_Gaz_LoLo_In AND (#Burn_Work OR #Burner.CMD_Start OR #Burner.CMD_Start_Stop) THEN
       #Burner.Alarm_W.%X5 := TRUE;
   END_IF;

   IF #P_Gaz_HiHi_In AND (#Burn_Work OR #Burner.CMD_Start OR #Burner.CMD_Start_Stop) THEN
       #Burner.Alarm_W.%X6 := TRUE;
   END_IF;

   IF #P_Gaz_LoLo AND (#Burn_Work OR #Burner.CMD_Start OR #Burner.CMD_Start_Stop) THEN
       #Burner.Alarm_W.%X7 := TRUE;
   END_IF;

   IF #P_Gaz_HiHi AND (#Burn_Work OR #Burner.CMD_Start OR #Burner.CMD_Start_Stop) THEN
       #Burner.Alarm_W.%X8 := TRUE;
   END_IF;

   IF #T_Emk_HiHi AND (#Burn_Work OR #Burner.CMD_Start OR #Burner.CMD_Start_Stop) THEN
       #Burner.Alarm_W.%X9 := TRUE;
   END_IF;

   IF #T_Oil_HiHi_Out AND (#Burn_Work OR #Burner.CMD_Start OR #Burner.CMD_Start_Stop) THEN
       #Burner.Alarm_W.%X10 := TRUE;
   END_IF;

   IF #Porog_2 THEN
       #Burner.Alarm_W.%X11 := TRUE;
   END_IF;

   IF #Valve_alarm_1 THEN
       #Burner.Alarm_W.%X12 := TRUE;
   END_IF;

   IF #Valve_alarm_2 THEN
       #Burner.Alarm_W.%X13 := TRUE;
   END_IF;

   IF #H_HiHi THEN
       #Burner.Alarm_W.%X14 := TRUE;
   END_IF;

   IF #H_LoLo THEN
       #Burner.Alarm_W.%X15 := TRUE;
   END_IF;

   IF #Burner.Alarm_W <> 0 THEN
       #Burner.Alarm := 1;
   END_IF;

   //пуск стоп горелки
   //Ручной режим (С панели)
   (*IF #Burner.mode = 0 THEN
       IF #Burner.CMD_Start AND NOT (#Burner.Alarm) THEN
           #Burner.CMD_Start_Stop := TRUE;
           #Burner.Fire := TRUE;
           #Need_open_cl_1 := TRUE;
       END_IF;
       IF #Burner.CMD_Stop OR #Burner.Alarm THEN
           #Burner.CMD_Start_Stop := FALSE;
           #Burner.Fire := FALSE;
           #Need_open_cl_1 := FALSE;
           #Need_open_cl_2 := FALSE;
           #Burner.Auto_Pause := FALSE;
           #Burner.CMD_Start := FALSE;
           #Burner.CMD_Stop := FALSE;
       END_IF;


       // Режим управления с АРМ    
   ELSIF #Burner.mode = 1 THEN
       IF #Burner.ARM_start AND NOT (#Burner.Alarm) THEN
           #Burner.CMD_Start_Stop := TRUE;
           #Burner.Fire := TRUE;
           #Need_open_cl_1 := TRUE;
       END_IF;
       IF #Burner.ARM_stop OR #Burner.Alarm THEN
           #Burner.CMD_Start_Stop := FALSE;
           #Burner.Fire := FALSE;
           #Need_open_cl_1 := FALSE;
           #Need_open_cl_2 := FALSE;
           #Burner.Auto_Pause := FALSE;
       END_IF;
   END_IF;*)
   "Delay_produv".TON(IN:=#Burner.CMD_Start_Stop,
                      PT:=T_CONV("DB_TST".Delay_produv)*1000);

   IF (#Burner.mode = 0 AND #Burner.CMD_Start) OR (#Burner.mode = 1 AND #Burner.ARM_start) OR (#Burner.Auto_Pause AND NOT #Burner.Flag_Auto_Pause) AND NOT (#Burner.Alarm) THEN
       #Burner.CMD_Start_Stop := TRUE;
   END_IF;
   IF #Burner.CMD_Start_Stop THEN
       #Burner.CMD_Start := FALSE;
       #Burner.ARM_start := FALSE;
       #Need_open_cl_1 := TRUE;
   END_IF;
   "Burner_Fire_Timer".TON(IN := #Need_open_cl_1 AND "Delay_produv".Q AND "EN",
                           PT := T_CONV("DB_TST".Fire_delay)*1000);
   IF #Need_open_cl_1 AND NOT #Burner.Fire AND NOT "Burner_Fire_Timer".Q AND "Delay_produv".Q AND NOT #Burn_Work AND #Burner.CMD_Start_Stop THEN
       #Burner.Fire := TRUE;
       "EN" := true;
   END_IF;
   "Burner_Fire_Timer_Delay".TON(IN := "Burner_Fire_Timer".Q,
                                 PT := T_CONV("DB_TST".Fire_interval)*1000);
   IF "Burner_Fire_Timer".Q THEN
       #Burner.Fire := false;
   END_IF;
   IF "Burner_Fire_Timer_Delay".Q THEN
       "EN" := FALSE;
   END_IF;
   "Start_Fire_Counter".CTU(CU:="Burner_Fire_Timer".Q,
                            R:=#Burner.Alarm OR #Burner.CMD_Stop OR #Burner.ARM_stop OR #Burn_Work,
                            PV:=3);
   IF "Start_Fire_Counter".QU THEN
       #Burner.Alarm_W.%X16 := TRUE;
   END_IF;
   IF (#Burner.mode = 0 AND #Burner.CMD_Stop) OR (#Burner.mode = 1 AND #Burner.ARM_stop) OR #Burner.Alarm THEN
       #Burner.CMD_Start_Stop := FALSE;
       #Burner.Fire := FALSE;
       #Need_open_cl_1 := FALSE;
       #Need_open_cl_2 := FALSE;
       #Burner.Auto_Pause := FALSE;
       #Burner.CMD_Start := FALSE;
       #Burner.CMD_Stop := FALSE;
   END_IF;

   //открытие клапана на основную горелку с задержкой по времени
   (*#Timer_need_cl_2.TON(IN := #Burn_Work,
                        PT := T#1s);*)
   (*IF #Burn_Work AND NOT (#Burner.Alarm) AND #Burner.CMD_Start_Stop THEN
       #Need_open_cl_2 := TRUE;
   END_IF;*)

   #Timer_need_cl_2.TON(IN := #Burn_Work AND NOT (#Burner.Alarm) AND #Burner.CMD_Start_Stop,
                        PT := T_CONV("DB_TST".Open_cl2_delay)*1000);

   IF #Timer_need_cl_2.Q THEN
       #Need_open_cl_2 := TRUE;
   END_IF;

   //авария по состоянию
   #Timer_Not_Start.TON(IN := #Burner.CMD_Start_Stop AND NOT(#Burner.Auto_Pause),
                        PT := T#1m);
   //игнорирование аварии при автопаузе
   IF #Timer_Not_Start.Q AND NOT (#Burn_Work) THEN
       IF NOT (#Burner.Auto_Pause) THEN
           #Burner.Alarm_W.%X16 := TRUE;
       END_IF;
   END_IF;

   // Если горелка горит и основной клапан открылся, то закрываем запальный клапан
   IF #Burn_Work AND "PLC_Signals_DB".DI_1_3.Output THEN
       #Need_open_cl_1 := FALSE;
   END_IF;

   //автопауза
   IF #Burner.CMD_Start_Stop AND
       (#T_Emk >= "DB_TST".T_Emk_Hi_Hmi OR #T_Oil >= "DB_TST".T_Oil_Hi_Hmi) AND NOT #Burner.Alarm THEN
           #Burner.Auto_Pause := TRUE;
           #Burner.Flag_Auto_Pause := TRUE;
           #Need_open_cl_1 := FALSE;
           #Need_open_cl_2 := FALSE;
           #Burner.CMD_Start_Stop := FALSE;
      (* ELSE
           #Burner.Flag_Auto_Pause := FALSE;*)
   END_IF;

   IF #Burner.Alarm THEN
       #Burner.Auto_Pause := FALSE;
       #Burner.Flag_Auto_Pause := FALSE;
   END_IF;

   //автопуск
    IF #Burner.Auto_Pause AND (#T_Emk <= "DB_TST".T_Emk_Lo_Hmi OR #T_Oil <= "DB_TST".T_Oil_Lo_Hmi) AND
        #Burner.Flag_Auto_Pause THEN
        #Burner.Flag_Auto_Pause := FALSE;
   END_IF;

   // Состояния горелки 
   IF (#Burner.Auto_Pause OR NOT #Burner.CMD_Start_Stop) AND NOT #Burner.Alarm  THEN
       #Burner.State := 0;
   ELSIF #Burner.CMD_Start_Stop AND NOT #Burner.Auto_Pause AND NOT #Burner.Alarm THEN
       #Burner.State := 1;
   ELSIF #Burner.Alarm THEN
       #Burner.State := 2;
   END_IF;



   IF #Burner.CMD_RST_Alarm OR #Burner.ARM_deblock THEN
       #Burner.Alarm_W := 0;
       #Burner.Alarm := FALSE;
   END_IF;
   #RST_Block_Burner := #Burner.CMD_RST_Alarm;

   IF #Burner.Fire THEN
       #Burner_fire := TRUE;
   ELSE
       #Burner_fire := FALSE;
   END_IF;

   IF #Burner.CMD_Start_Stop (*AND NOT (#Burner.Auto_Pause)*) THEN
       #Burner_ON := TRUE;
      // #Burner_fire := TRUE;
   ELSE
       #Burner_ON := FALSE;
       #Burner_fire := FALSE;
   END_IF;



   // Газоанализатор 
   "DB_TST".Gaz_porog1 := "PLC_Signals_DB".AI_2_6.State.%X2;
   "DB_TST".Gaz_porog2 := "PLC_Signals_DB".AI_2_6.State.%X1;
   "DB_TST".Gaz_neispravnost := "PLC_Signals_DB".AI_2_6.State.%X5;
END_FUNCTION

FUNCTION "AI_Config" : Void   // FC17, SCL
{ S7_Optimized_Access := 'TRUE' }
VERSION : 0.1
   VAR_INPUT
      Channel_Number : Int;
   END_VAR
   VAR_IN_OUT
      Config_AI : Struct
         Hihi_Value : Real;   // Уставка: Hihi
         High_Value : Real;   // Уставка: High
         Low_Value : Real;   // Уставка: Low
         Lolo_Value : Real;   // Уставка: Lolo
         MIN_Current : Real;   // Настройка: Минимальное входное значение тока
         MAX_Current : Real;   // Настройка: Максимальное входное значение тока
         MAX_Value : Real;   // Настройка: Максимальное значение измеряемой величины
         MIN_Value : Real;   // Настройка: Минимальное значение измеряемой величины
         Underflow_RAW : Real;   // Настройка: Значение кода ацп при обрыве
         Overflow_RAW : Real;   // Настройка: Значение кода ацп при зашкале
         SCALED : Real;   // Выход: Масштабированное в инженерные единицы значение входного сигнала
         ING_Value : Real;   // Выход: Токовое значение датчика
         Manual_Value : Real;   // Значение, введенное вручную
         Alarm_Delay : Int;   // Настройка: Задержка срабатывания аварий
         Warning_Delay : Int;   // Настройка: Задержка срабатывания предупреждений
         AVG_Delay : Real;   // Настройка: Зона нечувствительности
         Underflow_Delay : Int;   // Настройка: Задержка отображения обрыва датчика
         Overflow_Delay : Int;   // Настройка: Задержка отображения неисправности датчика
         StateHMI : Int;
         State : Word;   // Выход: Состояние датчика
         Modeee : Word;   // Настройка: Режим работы датчика
         bools : Word;   // Все булевы параметры AI
         AI_RAW_MIN : Int;   // Мин кода ацп
         AI_RAW_MAX : Int;   // Макс кода ацп
         Hihi_EN : Bool;   // Разрешение на сработку
         High_EN : Bool;   // Разрешение на сработку
         Low_En : Bool;   // Разрешение на сработку
         Lolo_EN : Bool;   // Разрешение на сработку
      END_STRUCT;
      AI_2_0 : Struct
         Hihi_Value : Real;   // Уставка: Hihi
         High_Value : Real;   // Уставка: High
         Low_Value : Real;   // Уставка: Low
         Lolo_Value : Real;   // Уставка: Lolo
         MIN_Current : Real;   // Настройка: Минимальное входное значение тока
         MAX_Current : Real;   // Настройка: Максимальное входное значение тока
         MAX_Value : Real;   // Настройка: Максимальное значение измеряемой величины
         MIN_Value : Real;   // Настройка: Минимальное значение измеряемой величины
         Underflow_RAW : Real;   // Настройка: Значение кода ацп при обрыве
         Overflow_RAW : Real;   // Настройка: Значение кода ацп при зашкале
         SCALED : Real;   // Выход: Масштабированное в инженерные единицы значение входного сигнала
         ING_Value : Real;   // Выход: Токовое значение датчика
         Manual_Value : Real;   // Значение, введенное вручную
         Alarm_Delay : Int;   // Настройка: Задержка срабатывания аварий
         Warning_Delay : Int;   // Настройка: Задержка срабатывания предупреждений
         AVG_Delay : Real;   // Настройка: Зона нечувствительности
         Underflow_Delay : Int;   // Настройка: Задержка отображения обрыва датчика
         Overflow_Delay : Int;   // Настройка: Задержка отображения неисправности датчика
         StateHMI : Int;
         State : Word;   // Выход: Состояние датчика
         Modeee : Word;   // Настройка: Режим работы датчика
         bools : Word;   // Все булевы параметры AI
         AI_RAW_MIN : Int;   // Мин кода ацп
         AI_RAW_MAX : Int;   // Макс кода ацп
         Hihi_EN : Bool;   // Разрешение на сработку
         High_EN : Bool;   // Разрешение на сработку
         Low_En : Bool;   // Разрешение на сработку
         Lolo_EN : Bool;   // Разрешение на сработку
      END_STRUCT;
      AI_2_1 : Struct
         Hihi_Value : Real;   // Уставка: Hihi
         High_Value : Real;   // Уставка: High
         Low_Value : Real;   // Уставка: Low
         Lolo_Value : Real;   // Уставка: Lolo
         MIN_Current : Real;   // Настройка: Минимальное входное значение тока
         MAX_Current : Real;   // Настройка: Максимальное входное значение тока
         MAX_Value : Real;   // Настройка: Максимальное значение измеряемой величины
         MIN_Value : Real;   // Настройка: Минимальное значение измеряемой величины
         Underflow_RAW : Real;   // Настройка: Значение кода ацп при обрыве
         Overflow_RAW : Real;   // Настройка: Значение кода ацп при зашкале
         SCALED : Real;   // Выход: Масштабированное в инженерные единицы значение входного сигнала
         ING_Value : Real;   // Выход: Токовое значение датчика
         Manual_Value : Real;   // Значение, введенное вручную
         Alarm_Delay : Int;   // Настройка: Задержка срабатывания аварий
         Warning_Delay : Int;   // Настройка: Задержка срабатывания предупреждений
         AVG_Delay : Real;   // Настройка: Зона нечувствительности
         Underflow_Delay : Int;   // Настройка: Задержка отображения обрыва датчика
         Overflow_Delay : Int;   // Настройка: Задержка отображения неисправности датчика
         StateHMI : Int;
         State : Word;   // Выход: Состояние датчика
         Modeee : Word;   // Настройка: Режим работы датчика
         bools : Word;   // Все булевы параметры AI
         AI_RAW_MIN : Int;   // Мин кода ацп
         AI_RAW_MAX : Int;   // Макс кода ацп
         Hihi_EN : Bool;   // Разрешение на сработку
         High_EN : Bool;   // Разрешение на сработку
         Low_En : Bool;   // Разрешение на сработку
         Lolo_EN : Bool;   // Разрешение на сработку
      END_STRUCT;
      AI_2_2 : Struct
         Hihi_Value : Real;   // Уставка: Hihi
         High_Value : Real;   // Уставка: High
         Low_Value : Real;   // Уставка: Low
         Lolo_Value : Real;   // Уставка: Lolo
         MIN_Current : Real;   // Настройка: Минимальное входное значение тока
         MAX_Current : Real;   // Настройка: Максимальное входное значение тока
         MAX_Value : Real;   // Настройка: Максимальное значение измеряемой величины
         MIN_Value : Real;   // Настройка: Минимальное значение измеряемой величины
         Underflow_RAW : Real;   // Настройка: Значение кода ацп при обрыве
         Overflow_RAW : Real;   // Настройка: Значение кода ацп при зашкале
         SCALED : Real;   // Выход: Масштабированное в инженерные единицы значение входного сигнала
         ING_Value : Real;   // Выход: Токовое значение датчика
         Manual_Value : Real;   // Значение, введенное вручную
         Alarm_Delay : Int;   // Настройка: Задержка срабатывания аварий
         Warning_Delay : Int;   // Настройка: Задержка срабатывания предупреждений
         AVG_Delay : Real;   // Настройка: Зона нечувствительности
         Underflow_Delay : Int;   // Настройка: Задержка отображения обрыва датчика
         Overflow_Delay : Int;   // Настройка: Задержка отображения неисправности датчика
         StateHMI : Int;
         State : Word;   // Выход: Состояние датчика
         Modeee : Word;   // Настройка: Режим работы датчика
         bools : Word;   // Все булевы параметры AI
         AI_RAW_MIN : Int;   // Мин кода ацп
         AI_RAW_MAX : Int;   // Макс кода ацп
         Hihi_EN : Bool;   // Разрешение на сработку
         High_EN : Bool;   // Разрешение на сработку
         Low_En : Bool;   // Разрешение на сработку
         Lolo_EN : Bool;   // Разрешение на сработку
      END_STRUCT;
      AI_2_3 : Struct
         Hihi_Value : Real;   // Уставка: Hihi
         High_Value : Real;   // Уставка: High
         Low_Value : Real;   // Уставка: Low
         Lolo_Value : Real;   // Уставка: Lolo
         MIN_Current : Real;   // Настройка: Минимальное входное значение тока
         MAX_Current : Real;   // Настройка: Максимальное входное значение тока
         MAX_Value : Real;   // Настройка: Максимальное значение измеряемой величины
         MIN_Value : Real;   // Настройка: Минимальное значение измеряемой величины
         Underflow_RAW : Real;   // Настройка: Значение кода ацп при обрыве
         Overflow_RAW : Real;   // Настройка: Значение кода ацп при зашкале
         SCALED : Real;   // Выход: Масштабированное в инженерные единицы значение входного сигнала
         ING_Value : Real;   // Выход: Токовое значение датчика
         Manual_Value : Real;   // Значение, введенное вручную
         Alarm_Delay : Int;   // Настройка: Задержка срабатывания аварий
         Warning_Delay : Int;   // Настройка: Задержка срабатывания предупреждений
         AVG_Delay : Real;   // Настройка: Зона нечувствительности
         Underflow_Delay : Int;   // Настройка: Задержка отображения обрыва датчика
         Overflow_Delay : Int;   // Настройка: Задержка отображения неисправности датчика
         StateHMI : Int;
         State : Word;   // Выход: Состояние датчика
         Modeee : Word;   // Настройка: Режим работы датчика
         bools : Word;   // Все булевы параметры AI
         AI_RAW_MIN : Int;   // Мин кода ацп
         AI_RAW_MAX : Int;   // Макс кода ацп
         Hihi_EN : Bool;   // Разрешение на сработку
         High_EN : Bool;   // Разрешение на сработку
         Low_En : Bool;   // Разрешение на сработку
         Lolo_EN : Bool;   // Разрешение на сработку
      END_STRUCT;
      AI_2_4 : Struct
         Hihi_Value : Real;   // Уставка: Hihi
         High_Value : Real;   // Уставка: High
         Low_Value : Real;   // Уставка: Low
         Lolo_Value : Real;   // Уставка: Lolo
         MIN_Current : Real;   // Настройка: Минимальное входное значение тока
         MAX_Current : Real;   // Настройка: Максимальное входное значение тока
         MAX_Value : Real;   // Настройка: Максимальное значение измеряемой величины
         MIN_Value : Real;   // Настройка: Минимальное значение измеряемой величины
         Underflow_RAW : Real;   // Настройка: Значение кода ацп при обрыве
         Overflow_RAW : Real;   // Настройка: Значение кода ацп при зашкале
         SCALED : Real;   // Выход: Масштабированное в инженерные единицы значение входного сигнала
         ING_Value : Real;   // Выход: Токовое значение датчика
         Manual_Value : Real;   // Значение, введенное вручную
         Alarm_Delay : Int;   // Настройка: Задержка срабатывания аварий
         Warning_Delay : Int;   // Настройка: Задержка срабатывания предупреждений
         AVG_Delay : Real;   // Настройка: Зона нечувствительности
         Underflow_Delay : Int;   // Настройка: Задержка отображения обрыва датчика
         Overflow_Delay : Int;   // Настройка: Задержка отображения неисправности датчика
         StateHMI : Int;
         State : Word;   // Выход: Состояние датчика
         Modeee : Word;   // Настройка: Режим работы датчика
         bools : Word;   // Все булевы параметры AI
         AI_RAW_MIN : Int;   // Мин кода ацп
         AI_RAW_MAX : Int;   // Макс кода ацп
         Hihi_EN : Bool;   // Разрешение на сработку
         High_EN : Bool;   // Разрешение на сработку
         Low_En : Bool;   // Разрешение на сработку
         Lolo_EN : Bool;   // Разрешение на сработку
      END_STRUCT;
      AI_2_5 : Struct
         Hihi_Value : Real;   // Уставка: Hihi
         High_Value : Real;   // Уставка: High
         Low_Value : Real;   // Уставка: Low
         Lolo_Value : Real;   // Уставка: Lolo
         MIN_Current : Real;   // Настройка: Минимальное входное значение тока
         MAX_Current : Real;   // Настройка: Максимальное входное значение тока
         MAX_Value : Real;   // Настройка: Максимальное значение измеряемой величины
         MIN_Value : Real;   // Настройка: Минимальное значение измеряемой величины
         Underflow_RAW : Real;   // Настройка: Значение кода ацп при обрыве
         Overflow_RAW : Real;   // Настройка: Значение кода ацп при зашкале
         SCALED : Real;   // Выход: Масштабированное в инженерные единицы значение входного сигнала
         ING_Value : Real;   // Выход: Токовое значение датчика
         Manual_Value : Real;   // Значение, введенное вручную
         Alarm_Delay : Int;   // Настройка: Задержка срабатывания аварий
         Warning_Delay : Int;   // Настройка: Задержка срабатывания предупреждений
         AVG_Delay : Real;   // Настройка: Зона нечувствительности
         Underflow_Delay : Int;   // Настройка: Задержка отображения обрыва датчика
         Overflow_Delay : Int;   // Настройка: Задержка отображения неисправности датчика
         StateHMI : Int;
         State : Word;   // Выход: Состояние датчика
         Modeee : Word;   // Настройка: Режим работы датчика
         bools : Word;   // Все булевы параметры AI
         AI_RAW_MIN : Int;   // Мин кода ацп
         AI_RAW_MAX : Int;   // Макс кода ацп
         Hihi_EN : Bool;   // Разрешение на сработку
         High_EN : Bool;   // Разрешение на сработку
         Low_En : Bool;   // Разрешение на сработку
         Lolo_EN : Bool;   // Разрешение на сработку
      END_STRUCT;
      AI_2_6 : Struct
         Hihi_Value : Real;   // Уставка: Hihi
         High_Value : Real;   // Уставка: High
         Low_Value : Real;   // Уставка: Low
         Lolo_Value : Real;   // Уставка: Lolo
         MIN_Current : Real;   // Настройка: Минимальное входное значение тока
         MAX_Current : Real;   // Настройка: Максимальное входное значение тока
         MAX_Value : Real;   // Настройка: Максимальное значение измеряемой величины
         MIN_Value : Real;   // Настройка: Минимальное значение измеряемой величины
         Underflow_RAW : Real;   // Настройка: Значение кода ацп при обрыве
         Overflow_RAW : Real;   // Настройка: Значение кода ацп при зашкале
         SCALED : Real;   // Выход: Масштабированное в инженерные единицы значение входного сигнала
         ING_Value : Real;   // Выход: Токовое значение датчика
         Manual_Value : Real;   // Значение, введенное вручную
         Alarm_Delay : Int;   // Настройка: Задержка срабатывания аварий
         Warning_Delay : Int;   // Настройка: Задержка срабатывания предупреждений
         AVG_Delay : Real;   // Настройка: Зона нечувствительности
         Underflow_Delay : Int;   // Настройка: Задержка отображения обрыва датчика
         Overflow_Delay : Int;   // Настройка: Задержка отображения неисправности датчика
         StateHMI : Int;
         State : Word;   // Выход: Состояние датчика
         Modeee : Word;   // Настройка: Режим работы датчика
         bools : Word;   // Все булевы параметры AI
         AI_RAW_MIN : Int;   // Мин кода ацп
         AI_RAW_MAX : Int;   // Макс кода ацп
         Hihi_EN : Bool;   // Разрешение на сработку
         High_EN : Bool;   // Разрешение на сработку
         Low_En : Bool;   // Разрешение на сработку
         Lolo_EN : Bool;   // Разрешение на сработку
      END_STRUCT;
      AI_2_7 : Struct
         Hihi_Value : Real;   // Уставка: Hihi
         High_Value : Real;   // Уставка: High
         Low_Value : Real;   // Уставка: Low
         Lolo_Value : Real;   // Уставка: Lolo
         MIN_Current : Real;   // Настройка: Минимальное входное значение тока
         MAX_Current : Real;   // Настройка: Максимальное входное значение тока
         MAX_Value : Real;   // Настройка: Максимальное значение измеряемой величины
         MIN_Value : Real;   // Настройка: Минимальное значение измеряемой величины
         Underflow_RAW : Real;   // Настройка: Значение кода ацп при обрыве
         Overflow_RAW : Real;   // Настройка: Значение кода ацп при зашкале
         SCALED : Real;   // Выход: Масштабированное в инженерные единицы значение входного сигнала
         ING_Value : Real;   // Выход: Токовое значение датчика
         Manual_Value : Real;   // Значение, введенное вручную
         Alarm_Delay : Int;   // Настройка: Задержка срабатывания аварий
         Warning_Delay : Int;   // Настройка: Задержка срабатывания предупреждений
         AVG_Delay : Real;   // Настройка: Зона нечувствительности
         Underflow_Delay : Int;   // Настройка: Задержка отображения обрыва датчика
         Overflow_Delay : Int;   // Настройка: Задержка отображения неисправности датчика
         StateHMI : Int;
         State : Word;   // Выход: Состояние датчика
         Modeee : Word;   // Настройка: Режим работы датчика
         bools : Word;   // Все булевы параметры AI
         AI_RAW_MIN : Int;   // Мин кода ацп
         AI_RAW_MAX : Int;   // Макс кода ацп
         Hihi_EN : Bool;   // Разрешение на сработку
         High_EN : Bool;   // Разрешение на сработку
         Low_En : Bool;   // Разрешение на сработку
         Lolo_EN : Bool;   // Разрешение на сработку
      END_STRUCT;
      AI_3_0 : Struct
         Hihi_Value : Real;   // Уставка: Hihi
         High_Value : Real;   // Уставка: High
         Low_Value : Real;   // Уставка: Low
         Lolo_Value : Real;   // Уставка: Lolo
         MIN_Current : Real;   // Настройка: Минимальное входное значение тока
         MAX_Current : Real;   // Настройка: Максимальное входное значение тока
         MAX_Value : Real;   // Настройка: Максимальное значение измеряемой величины
         MIN_Value : Real;   // Настройка: Минимальное значение измеряемой величины
         Underflow_RAW : Real;   // Настройка: Значение кода ацп при обрыве
         Overflow_RAW : Real;   // Настройка: Значение кода ацп при зашкале
         SCALED : Real;   // Выход: Масштабированное в инженерные единицы значение входного сигнала
         ING_Value : Real;   // Выход: Токовое значение датчика
         Manual_Value : Real;   // Значение, введенное вручную
         Alarm_Delay : Int;   // Настройка: Задержка срабатывания аварий
         Warning_Delay : Int;   // Настройка: Задержка срабатывания предупреждений
         AVG_Delay : Real;   // Настройка: Зона нечувствительности
         Underflow_Delay : Int;   // Настройка: Задержка отображения обрыва датчика
         Overflow_Delay : Int;   // Настройка: Задержка отображения неисправности датчика
         StateHMI : Int;
         State : Word;   // Выход: Состояние датчика
         Modeee : Word;   // Настройка: Режим работы датчика
         bools : Word;   // Все булевы параметры AI
         AI_RAW_MIN : Int;   // Мин кода ацп
         AI_RAW_MAX : Int;   // Макс кода ацп
         Hihi_EN : Bool;   // Разрешение на сработку
         High_EN : Bool;   // Разрешение на сработку
         Low_En : Bool;   // Разрешение на сработку
         Lolo_EN : Bool;   // Разрешение на сработку
      END_STRUCT;
      AI_3_1 : Struct
         Hihi_Value : Real;   // Уставка: Hihi
         High_Value : Real;   // Уставка: High
         Low_Value : Real;   // Уставка: Low
         Lolo_Value : Real;   // Уставка: Lolo
         MIN_Current : Real;   // Настройка: Минимальное входное значение тока
         MAX_Current : Real;   // Настройка: Максимальное входное значение тока
         MAX_Value : Real;   // Настройка: Максимальное значение измеряемой величины
         MIN_Value : Real;   // Настройка: Минимальное значение измеряемой величины
         Underflow_RAW : Real;   // Настройка: Значение кода ацп при обрыве
         Overflow_RAW : Real;   // Настройка: Значение кода ацп при зашкале
         SCALED : Real;   // Выход: Масштабированное в инженерные единицы значение входного сигнала
         ING_Value : Real;   // Выход: Токовое значение датчика
         Manual_Value : Real;   // Значение, введенное вручную
         Alarm_Delay : Int;   // Настройка: Задержка срабатывания аварий
         Warning_Delay : Int;   // Настройка: Задержка срабатывания предупреждений
         AVG_Delay : Real;   // Настройка: Зона нечувствительности
         Underflow_Delay : Int;   // Настройка: Задержка отображения обрыва датчика
         Overflow_Delay : Int;   // Настройка: Задержка отображения неисправности датчика
         StateHMI : Int;
         State : Word;   // Выход: Состояние датчика
         Modeee : Word;   // Настройка: Режим работы датчика
         bools : Word;   // Все булевы параметры AI
         AI_RAW_MIN : Int;   // Мин кода ацп
         AI_RAW_MAX : Int;   // Макс кода ацп
         Hihi_EN : Bool;   // Разрешение на сработку
         High_EN : Bool;   // Разрешение на сработку
         Low_En : Bool;   // Разрешение на сработку
         Lolo_EN : Bool;   // Разрешение на сработку
      END_STRUCT;
      AI_3_2 : Struct
         Hihi_Value : Real;   // Уставка: Hihi
         High_Value : Real;   // Уставка: High
         Low_Value : Real;   // Уставка: Low
         Lolo_Value : Real;   // Уставка: Lolo
         MIN_Current : Real;   // Настройка: Минимальное входное значение тока
         MAX_Current : Real;   // Настройка: Максимальное входное значение тока
         MAX_Value : Real;   // Настройка: Максимальное значение измеряемой величины
         MIN_Value : Real;   // Настройка: Минимальное значение измеряемой величины
         Underflow_RAW : Real;   // Настройка: Значение кода ацп при обрыве
         Overflow_RAW : Real;   // Настройка: Значение кода ацп при зашкале
         SCALED : Real;   // Выход: Масштабированное в инженерные единицы значение входного сигнала
         ING_Value : Real;   // Выход: Токовое значение датчика
         Manual_Value : Real;   // Значение, введенное вручную
         Alarm_Delay : Int;   // Настройка: Задержка срабатывания аварий
         Warning_Delay : Int;   // Настройка: Задержка срабатывания предупреждений
         AVG_Delay : Real;   // Настройка: Зона нечувствительности
         Underflow_Delay : Int;   // Настройка: Задержка отображения обрыва датчика
         Overflow_Delay : Int;   // Настройка: Задержка отображения неисправности датчика
         StateHMI : Int;
         State : Word;   // Выход: Состояние датчика
         Modeee : Word;   // Настройка: Режим работы датчика
         bools : Word;   // Все булевы параметры AI
         AI_RAW_MIN : Int;   // Мин кода ацп
         AI_RAW_MAX : Int;   // Макс кода ацп
         Hihi_EN : Bool;   // Разрешение на сработку
         High_EN : Bool;   // Разрешение на сработку
         Low_En : Bool;   // Разрешение на сработку
         Lolo_EN : Bool;   // Разрешение на сработку
      END_STRUCT;
      AI_3_3 : Struct
         Hihi_Value : Real;   // Уставка: Hihi
         High_Value : Real;   // Уставка: High
         Low_Value : Real;   // Уставка: Low
         Lolo_Value : Real;   // Уставка: Lolo
         MIN_Current : Real;   // Настройка: Минимальное входное значение тока
         MAX_Current : Real;   // Настройка: Максимальное входное значение тока
         MAX_Value : Real;   // Настройка: Максимальное значение измеряемой величины
         MIN_Value : Real;   // Настройка: Минимальное значение измеряемой величины
         Underflow_RAW : Real;   // Настройка: Значение кода ацп при обрыве
         Overflow_RAW : Real;   // Настройка: Значение кода ацп при зашкале
         SCALED : Real;   // Выход: Масштабированное в инженерные единицы значение входного сигнала
         ING_Value : Real;   // Выход: Токовое значение датчика
         Manual_Value : Real;   // Значение, введенное вручную
         Alarm_Delay : Int;   // Настройка: Задержка срабатывания аварий
         Warning_Delay : Int;   // Настройка: Задержка срабатывания предупреждений
         AVG_Delay : Real;   // Настройка: Зона нечувствительности
         Underflow_Delay : Int;   // Настройка: Задержка отображения обрыва датчика
         Overflow_Delay : Int;   // Настройка: Задержка отображения неисправности датчика
         StateHMI : Int;
         State : Word;   // Выход: Состояние датчика
         Modeee : Word;   // Настройка: Режим работы датчика
         bools : Word;   // Все булевы параметры AI
         AI_RAW_MIN : Int;   // Мин кода ацп
         AI_RAW_MAX : Int;   // Макс кода ацп
         Hihi_EN : Bool;   // Разрешение на сработку
         High_EN : Bool;   // Разрешение на сработку
         Low_En : Bool;   // Разрешение на сработку
         Lolo_EN : Bool;   // Разрешение на сработку
      END_STRUCT;
      AI_3_4 : Struct
         Hihi_Value : Real;   // Уставка: Hihi
         High_Value : Real;   // Уставка: High
         Low_Value : Real;   // Уставка: Low
         Lolo_Value : Real;   // Уставка: Lolo
         MIN_Current : Real;   // Настройка: Минимальное входное значение тока
         MAX_Current : Real;   // Настройка: Максимальное входное значение тока
         MAX_Value : Real;   // Настройка: Максимальное значение измеряемой величины
         MIN_Value : Real;   // Настройка: Минимальное значение измеряемой величины
         Underflow_RAW : Real;   // Настройка: Значение кода ацп при обрыве
         Overflow_RAW : Real;   // Настройка: Значение кода ацп при зашкале
         SCALED : Real;   // Выход: Масштабированное в инженерные единицы значение входного сигнала
         ING_Value : Real;   // Выход: Токовое значение датчика
         Manual_Value : Real;   // Значение, введенное вручную
         Alarm_Delay : Int;   // Настройка: Задержка срабатывания аварий
         Warning_Delay : Int;   // Настройка: Задержка срабатывания предупреждений
         AVG_Delay : Real;   // Настройка: Зона нечувствительности
         Underflow_Delay : Int;   // Настройка: Задержка отображения обрыва датчика
         Overflow_Delay : Int;   // Настройка: Задержка отображения неисправности датчика
         StateHMI : Int;
         State : Word;   // Выход: Состояние датчика
         Modeee : Word;   // Настройка: Режим работы датчика
         bools : Word;   // Все булевы параметры AI
         AI_RAW_MIN : Int;   // Мин кода ацп
         AI_RAW_MAX : Int;   // Макс кода ацп
         Hihi_EN : Bool;   // Разрешение на сработку
         High_EN : Bool;   // Разрешение на сработку
         Low_En : Bool;   // Разрешение на сработку
         Lolo_EN : Bool;   // Разрешение на сработку
      END_STRUCT;
      AI_3_5 : Struct
         Hihi_Value : Real;   // Уставка: Hihi
         High_Value : Real;   // Уставка: High
         Low_Value : Real;   // Уставка: Low
         Lolo_Value : Real;   // Уставка: Lolo
         MIN_Current : Real;   // Настройка: Минимальное входное значение тока
         MAX_Current : Real;   // Настройка: Максимальное входное значение тока
         MAX_Value : Real;   // Настройка: Максимальное значение измеряемой величины
         MIN_Value : Real;   // Настройка: Минимальное значение измеряемой величины
         Underflow_RAW : Real;   // Настройка: Значение кода ацп при обрыве
         Overflow_RAW : Real;   // Настройка: Значение кода ацп при зашкале
         SCALED : Real;   // Выход: Масштабированное в инженерные единицы значение входного сигнала
         ING_Value : Real;   // Выход: Токовое значение датчика
         Manual_Value : Real;   // Значение, введенное вручную
         Alarm_Delay : Int;   // Настройка: Задержка срабатывания аварий
         Warning_Delay : Int;   // Настройка: Задержка срабатывания предупреждений
         AVG_Delay : Real;   // Настройка: Зона нечувствительности
         Underflow_Delay : Int;   // Настройка: Задержка отображения обрыва датчика
         Overflow_Delay : Int;   // Настройка: Задержка отображения неисправности датчика
         StateHMI : Int;
         State : Word;   // Выход: Состояние датчика
         Modeee : Word;   // Настройка: Режим работы датчика
         bools : Word;   // Все булевы параметры AI
         AI_RAW_MIN : Int;   // Мин кода ацп
         AI_RAW_MAX : Int;   // Макс кода ацп
         Hihi_EN : Bool;   // Разрешение на сработку
         High_EN : Bool;   // Разрешение на сработку
         Low_En : Bool;   // Разрешение на сработку
         Lolo_EN : Bool;   // Разрешение на сработку
      END_STRUCT;
      AI_3_6 : Struct
         Hihi_Value : Real;   // Уставка: Hihi
         High_Value : Real;   // Уставка: High
         Low_Value : Real;   // Уставка: Low
         Lolo_Value : Real;   // Уставка: Lolo
         MIN_Current : Real;   // Настройка: Минимальное входное значение тока
         MAX_Current : Real;   // Настройка: Максимальное входное значение тока
         MAX_Value : Real;   // Настройка: Максимальное значение измеряемой величины
         MIN_Value : Real;   // Настройка: Минимальное значение измеряемой величины
         Underflow_RAW : Real;   // Настройка: Значение кода ацп при обрыве
         Overflow_RAW : Real;   // Настройка: Значение кода ацп при зашкале
         SCALED : Real;   // Выход: Масштабированное в инженерные единицы значение входного сигнала
         ING_Value : Real;   // Выход: Токовое значение датчика
         Manual_Value : Real;   // Значение, введенное вручную
         Alarm_Delay : Int;   // Настройка: Задержка срабатывания аварий
         Warning_Delay : Int;   // Настройка: Задержка срабатывания предупреждений
         AVG_Delay : Real;   // Настройка: Зона нечувствительности
         Underflow_Delay : Int;   // Настройка: Задержка отображения обрыва датчика
         Overflow_Delay : Int;   // Настройка: Задержка отображения неисправности датчика
         StateHMI : Int;
         State : Word;   // Выход: Состояние датчика
         Modeee : Word;   // Настройка: Режим работы датчика
         bools : Word;   // Все булевы параметры AI
         AI_RAW_MIN : Int;   // Мин кода ацп
         AI_RAW_MAX : Int;   // Макс кода ацп
         Hihi_EN : Bool;   // Разрешение на сработку
         High_EN : Bool;   // Разрешение на сработку
         Low_En : Bool;   // Разрешение на сработку
         Lolo_EN : Bool;   // Разрешение на сработку
      END_STRUCT;
      AI_3_7 : Struct
         Hihi_Value : Real;   // Уставка: Hihi
         High_Value : Real;   // Уставка: High
         Low_Value : Real;   // Уставка: Low
         Lolo_Value : Real;   // Уставка: Lolo
         MIN_Current : Real;   // Настройка: Минимальное входное значение тока
         MAX_Current : Real;   // Настройка: Максимальное входное значение тока
         MAX_Value : Real;   // Настройка: Максимальное значение измеряемой величины
         MIN_Value : Real;   // Настройка: Минимальное значение измеряемой величины
         Underflow_RAW : Real;   // Настройка: Значение кода ацп при обрыве
         Overflow_RAW : Real;   // Настройка: Значение кода ацп при зашкале
         SCALED : Real;   // Выход: Масштабированное в инженерные единицы значение входного сигнала
         ING_Value : Real;   // Выход: Токовое значение датчика
         Manual_Value : Real;   // Значение, введенное вручную
         Alarm_Delay : Int;   // Настройка: Задержка срабатывания аварий
         Warning_Delay : Int;   // Настройка: Задержка срабатывания предупреждений
         AVG_Delay : Real;   // Настройка: Зона нечувствительности
         Underflow_Delay : Int;   // Настройка: Задержка отображения обрыва датчика
         Overflow_Delay : Int;   // Настройка: Задержка отображения неисправности датчика
         StateHMI : Int;
         State : Word;   // Выход: Состояние датчика
         Modeee : Word;   // Настройка: Режим работы датчика
         bools : Word;   // Все булевы параметры AI
         AI_RAW_MIN : Int;   // Мин кода ацп
         AI_RAW_MAX : Int;   // Макс кода ацп
         Hihi_EN : Bool;   // Разрешение на сработку
         High_EN : Bool;   // Разрешение на сработку
         Low_En : Bool;   // Разрешение на сработку
         Lolo_EN : Bool;   // Разрешение на сработку
      END_STRUCT;
      Read : Bool;
      Write : Bool;
   END_VAR
BEGIN
   IF "PLC_Signals_DB".CH_NUMBER[1] THEN
       "DB_TST".CH_NUMBER := 1;
   END_IF;
   IF "PLC_Signals_DB".CH_NUMBER[2] THEN
       "DB_TST".CH_NUMBER := 2;
   END_IF;
   IF "PLC_Signals_DB".CH_NUMBER[3] THEN
       "DB_TST".CH_NUMBER := 3;
   END_IF;
   IF "PLC_Signals_DB".CH_NUMBER[4] THEN
       "DB_TST".CH_NUMBER := 4;
   END_IF;
   IF "PLC_Signals_DB".CH_NUMBER[5] THEN
       "DB_TST".CH_NUMBER := 5;
   END_IF;
   IF "PLC_Signals_DB".CH_NUMBER[6] THEN
       "DB_TST".CH_NUMBER := 6;
   END_IF;
   IF "PLC_Signals_DB".CH_NUMBER[7] THEN
       "DB_TST".CH_NUMBER := 7;
   END_IF;
   IF "PLC_Signals_DB".CH_NUMBER[8] THEN
       "DB_TST".CH_NUMBER := 8;
   END_IF;
   IF "PLC_Signals_DB".CH_NUMBER[9] THEN
       "DB_TST".CH_NUMBER := 9;
   END_IF;
   IF "PLC_Signals_DB".CH_NUMBER[10] THEN
       "DB_TST".CH_NUMBER := 10;
   END_IF;
   IF "PLC_Signals_DB".CH_NUMBER[11] THEN
       "DB_TST".CH_NUMBER := 11;
   END_IF;
   IF "PLC_Signals_DB".CH_NUMBER[12] THEN
       "DB_TST".CH_NUMBER := 12;
   END_IF;
   IF "PLC_Signals_DB".CH_NUMBER[13] THEN
       "DB_TST".CH_NUMBER := 13;
   END_IF;
   IF "PLC_Signals_DB".CH_NUMBER[14] THEN
       "DB_TST".CH_NUMBER := 14;
   END_IF;
   IF "PLC_Signals_DB".CH_NUMBER[15] THEN
       "DB_TST".CH_NUMBER := 15;
   END_IF;
   IF "PLC_Signals_DB".CH_NUMBER[16] THEN
       "DB_TST".CH_NUMBER := 16;
   END_IF;
   IF "PLC_Signals_DB".CH_NUMBER[17] THEN
       "DB_TST".CH_NUMBER := 17;
   END_IF;
   IF "PLC_Signals_DB".CH_NUMBER[18] THEN
       "DB_TST".CH_NUMBER := 18;
   END_IF;
   IF "PLC_Signals_DB".CH_NUMBER[19] THEN
       "DB_TST".CH_NUMBER := 19;
   END_IF;
   IF "PLC_Signals_DB".CH_NUMBER[20] THEN
       "DB_TST".CH_NUMBER := 20;
   END_IF;

